		CompressServo.fPosition:= 0;
		CompressServo.fVelocity:= 10; //mm/s
	
		CompressServo.xMoveA:=TRUE;
		StateNext:=5;
	5:	
		IF CompressServo.xInPosition = TRUE THEN
		
			CompressServo.xMoveA := FALSE;
			StateNext:=0;
			axis_ready:=TRUE;
		
		END_IF


	END_CASE

	State:=StateNext;
ELSIF NOT enable THEN
	axis_ready:=FALSE;
	CompressServo.xMoveA := FALSE;
	state:=0;
END_IF
END_METHOD

METHOD _Halt : BOOL
VAR_INPUT
END_VAR
CompressServo.xHalt:=TRUE;
END_METHOD

METHOD _Halt_false : BOOL
VAR_INPUT
END_VAR
CompressServo.xHalt:=FALSE;
END_METHOD

METHOD _Home : BOOL
VAR_INPUT
	
END_VAR


VAR

	
	
END_VAR

VAR_OUTPUT
	
END_VAR
CASE State OF //you are here

0:	
	_ExecutedHome := FALSE;
	CompressServo.fVelocity := ToolPositioningSpeed;
	CompressServo.fAxisAcceleration := ToolPositioningAccel;
	CompressServo.fAxisDeceleration := ToolPositioningAccel;
	CompressServo.fAxisJerk := ToolPositioningJerk;

	IF ixCompressHomeSwitch THEN
		CompressServo.xPositiveDirection := FALSE;
		IF  tickcounter_compress < 10 THEN
			tickcounter_compress := tickcounter_compress + 1;  // can be put in onditional
		
		ELSE
		//IF tickcounter_compress >= 10 THEN
			CompressServo.xMoveV := TRUE;
		END_IF
	ELSE
	
		//CompressServo.xHalt := NOT CompressServo.xHalt;
		CompressServo.xMoveV := FALSE;
		//CompressServo.xHalt := NOT CompressServo.xHalt;
		CompressServo.xHalt := TRUE;
		IF CompressServo.xHalted THEN
			tickcounter_compress:=0;
			StateNext := 5;
		END_IF
	
	END_IF
	
5:
	
	CompressServo.xHalt := FALSE;
	tickcounter_compress := tickcounter_compress + 1;
	IF tickcounter_compress >= 10 THEN
		tickcounter_compress := 0;
		StateNext := 10;
	END_IF
	
10:
	CompressServo.fVelocity := ToolHomingSpeed;
	
	IF NOT ixCompressHomeSwitch THEN
		CompressServo.xPositiveDirection := TRUE;
		IF tickcounter_compress < 10 THEN
			tickcounter_compress := tickcounter_compress + 1;
		ELSE
		//IF tickcounter >= 10 THEN
			CompressServo.xMoveV := TRUE;
		END_IF
	ELSE
		CompressServo.xMoveV := FALSE;
		CompressServo.xHalt := TRUE;
		IF CompressServo.xHalted AND CompressServo.fstandstill THEN
			tickcounter_compress := 0;
			StateNext := 15;
		END_IF
	END_IF

15:
	
	CompressServo.xHalt := FALSE;
	tickcounter_compress := tickcounter_compress + 1;
	IF tickcounter_compress >= 25 THEN
		tickcounter_compress := 0;
		StateNext := 20;
		//Executed := TRUE;
	END_IF	

20:
	CompressServo.fHomeOffset := 0;
	CompressServo.xZero := TRUE;
	StateNext := 25;	
	
25:
	IF CompressServo.xZeroed THEN
		CompressServo.xZero := FALSE;
		_ExecutedHome := TRUE;
		StateNext := 0;
	END_IF

END_CASE

State := StateNext;
END_METHOD

METHOD _Home_without_resetting : BOOL
VAR_INPUT
	enable			:BOOL;
END_VAR


VAR

	
	
END_VAR

VAR_OUTPUT
	
END_VAR

IF enable AND NOT axis_ready THEN
	CASE State OF //you are here

	0:	
		//_ExecutedHome := FALSE;
		CompressServo.fVelocity := ToolPositioningSpeed;
		CompressServo.fAxisAcceleration := ToolPositioningAccel;
		CompressServo.fAxisDeceleration := ToolPositioningAccel;
		CompressServo.fAxisJerk := ToolPositioningJerk;

		IF ixCompressHomeSwitch THEN
			CompressServo.xPositiveDirection := FALSE;
			//IF  tickcounter_compress < 10 THEN
			//	tickcounter_compress := tickcounter_compress + 1;  // can be put in onditional
		
			//ELSE
			//IF tickcounter_compress >= 10 THEN
			CompressServo.xMoveV := TRUE;
			//END_IF
		ELSE
	
			//CompressServo.xHalt := NOT CompressServo.xHalt;
			CompressServo.xMoveV := FALSE;
			//CompressServo.xHalt := NOT CompressServo.xHalt;
			CompressServo.xHalt := TRUE;
			statenext:=5;

	
		END_IF	
	5:
	
		IF CompressServo.xHalted THEN
			//tickcounter_compress:=0;
			CompressServo.xHalt := FALSE;
			StateNext := 10;
		END_IF
	
	10:
		CompressServo.fVelocity := ToolHomingSpeed;
	
		IF NOT ixCompressHomeSwitch THEN
			CompressServo.xPositiveDirection := TRUE;
			//IF tickcounter_compress < 10 THEN
			//	tickcounter_compress := tickcounter_compress + 1;
			//ELSE
			//IF tickcounter >= 10 THEN
			CompressServo.xMoveV := TRUE;
			//END_IF
		ELSE
			CompressServo.xMoveV := FALSE;
			CompressServo.xHalt := TRUE;
			IF CompressServo.xHalted AND CompressServo.fstandstill THEN
				tickcounter_compress := 0;
				StateNext := 15;
			END_IF
		END_IF

	15:
	
		CompressServo.xHalt := FALSE;
		tickcounter_compress := tickcounter_compress + 1;
		IF tickcounter_compress >= 25 THEN
			tickcounter_compress := 0;
			StateNext := 20;
			//Executed := TRUE;
		END_IF	

	20:

		//CompressServo.xZero := FALSE;
		axis_ready := TRUE;
		StateNext := 0;
	

	END_CASE

	State := StateNext;

ELSIF enable = FALSE THEN
	axis_ready:=FALSE;
	CompressServo.xHalt:=FALSE;
	CompressServo.xMoveV:=FALSE;
	state:=0;
	statenext:=0;
END_IF
END_METHOD

METHOD _manuel : BOOL
VAR_INPUT
	enable			:BOOL;
END_VAR
IF enable THEN
	IF NOT compress_settings.minus AND compress_settings.plus (*AND compressservo.xHalted*) THEN
		//CompressServo.xMoveV:=TRUE;
		Compressservo.fVelocity:=compress_settings.speed;
		CompressServo.xPositiveDirection := TRUE;
		CompressServo.xMoveV:=TRUE;
		CompressServo.xHalt:=FALSE;
	
	ELSIF NOT compress_settings.plus AND compress_settings.minus (*AND compressservo.xHalted*) THEN
	
		Compressservo.fVelocity:=compress_settings.speed;
		CompressServo.xPositiveDirection := FALSE;
		CompressServo.xMoveV:=TRUE;
		CompressServo.xHalt:=FALSE;	
	
	ELSIF NOT compress_settings.plus AND NOT compress_settings.minus THEN
	
		CompressServo.xHalt:=TRUE;
		CompressServo.xMoveV:=FALSE;
	
	END_IF
ELSE
	CompressServo.xHalt:=FALSE;
	CompressServo.xMoveV:=FALSE;
END_IF
END_METHOD

METHOD _mc_stop : BOOL
VAR_INPUT
END_VAR
CompressServo.xStop:=TRUE;
END_METHOD

METHOD _Reset
VAR_INPUT
END_VAR
	tickcounter_Compress:=0;
	CompressServoEnable := FALSE;
	CompressServo.xZero := FALSE;
	CompressServo.xMoveV := FALSE;
	CompressServo.xMoveA := FALSE;
	CompressServo.xHalt := FALSE;
	CompressServo.GearIn := FALSE;
	CompressServo.xStop:=FALSE;
	state:=0;
	statenext:=0;
	
	
	axis_ready:=FALSE;
	_ExecutedHome:=FALSE;
	_ExecutedOffset:=FALSE;
	PRG_Machine.reset_rec_old();
	PRG_Machine._debug(enable:=FALSE);
END_METHOD

METHOD _Reset_medium
VAR_INPUT
END_VAR
	tickcounter_Compress:=0;
	CompressServoEnable := FALSE;
	CompressServo.xZero := FALSE;
	CompressServo.xMoveV := FALSE;
	CompressServo.xMoveA := FALSE;
	CompressServo.xHalt := FALSE;
	CompressServo.GearIn := FALSE;
	CompressServo.xStop:=FALSE;
	state:=0;
	statenext:=0;
	
	
	axis_ready:=FALSE;
	PRG_Machine._debug(enable:=FALSE);
END_METHOD

METHOD _retract  : BOOL
VAR_INPUT
	Enable				:BOOL;
	
END_VAR
IF enable AND NOT axis_ready THEN
	CASE State OF
	
	0:	
	
		CompressServo.fPosition:= 0;
		CompressServo.fVelocity:= _Compress_Param.Pusher.Retract_Speed; //mm/s
	
		CompressServo.xMoveA:=TRUE;
		StateNext:=5;
	5:	
		IF CompressServo.xInPosition = TRUE THEN
		
			CompressServo.xMoveA := FALSE;
			StateNext:=0;
			axis_ready:=TRUE;
		
		END_IF


	END_CASE

	State:=StateNext;
ELSIF NOT enable THEN
	axis_ready:=FALSE;
	CompressServo.xMoveA := FALSE;
	state:=0;
END_IF
END_METHOD

METHOD _Soft_Reset
VAR_INPUT
END_VAR

tickcounter_Compress:=0;
CompressServo.xZero := FALSE;
CompressServo.xMoveV := FALSE;
CompressServo.xMoveA := FALSE;
CompressServo.xHalt := FALSE;
CompressServo.GearIn := FALSE;
CompressServo.xStop:=FALSE;
state:=0;
statenext:=0;

axis_ready:=FALSE;
PRG_Machine._debug(enable:=FALSE);
END_METHOD

METHOD _Update
VAR_INPUT
END_VAR
CompressServo(
	xEnable:= CompressServoEnable, 
	xZero:= , 
	xMoveR:= , 
	xMoveA:= , 
	xMoveV:= , 
	xPositiveDirection:= , 
	fDistance:= , 
	fPosition:= , 
	fVelocity:= , 
	xStop:= , 
	xHome:= , 
	xHomeFlag:= , 
	homePosition:=0,
	fActualPosition=> , 
	fActualVelocity=> , 
	fActModuloPos=> , 
	xEnabled=> CompressServoEnabled, 
	xMoveComplete=> , 
	xInPosition=> , 
	xAtSpeed=> , 
	xStopped=> , 
	xHomed=> ,
	errorID=> CompressServoErrorID, 
	Axis:= CompressAxis );
END_METHOD

PROPERTY Compress_Param : recipe
GET
Compress_param := _Compress_Param;
END_GET
SET
_Compress_param := Compress_Param;
END_SET
END_PROPERTY

PROPERTY HomeExecuted : BOOL
GET
HomeExecuted := _ExecutedHome;
END_GET
SET
_ExecutedHome := HomeExecuted;
END_SET
END_PROPERTY

METHOD Offset
VAR_INPUT
	Enable				:BOOL;
END_VAR

IF enable AND NOT axis_ready THEN	
	CASE State OF
	0:	
		_ExecutedOffset:=FALSE;
		CompressServo.fPosition:= _Compress_Param.Other.Compress_Home_Offset - PRG_Machine.rec_old.other.Compress_home_offset;
		CompressServo.fVelocity:= 20; //mm/s
	
		IF CompressServo.fPosition<>0 THEN
			CompressServo.xMoveA:=TRUE;
			StateNext:=5;
		ELSE
			_ExecutedOffset:=TRUE;
		END_IF
	
		//StateNext:=5;
	5:	
		IF CompressServo.xInPosition AND compressservo.fstandstill = TRUE THEN
			
			CompressServo.xMoveA := FALSE;
			StateNext:=7;
			//_ExecutedOffset:=TRUE;
		
		END_IF
	
	7:

		tickcounter_compress := tickcounter_compress + 1;
		IF tickcounter_compress >= 25 THEN
			tickcounter_compress := 0;
			StateNext := 10;
			//Executed := TRUE;
		END_IF	
	
	10:
	
		compressServo.fHomeOffset := 0;
		compressServo.xZero := TRUE;
		StateNext := 15;	
	
	15:
		IF compressServo.xZeroed THEN
			compressServo.xZero := FALSE;
			_ExecutedOffset:=TRUE;
			axis_ready:=TRUE;
			StateNext := 0;
		END_IF

	END_CASE

	State:=StateNext;
	
ELSIF NOT enable THEN 
	axis_ready:=FALSE;
	compressServo.xZero := FALSE;
	StateNext := 0;
END_IF
END_METHOD

PROPERTY OffsetExecuted : BOOL
GET
OffsetExecuted := _ExecutedOffset;
END_GET
SET
_ExecutedOffset := OffsetExecuted;
END_SET
END_PROPERTY

PROPERTY Stage1Executed : BOOL
GET
Stage1Executed := _ExecutedStage1;
END_GET
SET
_ExecutedStage1 := Stage1Executed;
END_SET
END_PROPERTY

PROPERTY Stage5Executed : BOOL
GET
Stage5Executed := _ExecutedStage5;
END_GET
SET
_ExecutedStage5 := Stage5Executed;
END_SET
END_PROPERTY

END_FUNCTION_BLOCK

// ---- Classes/Shield/FB_Shield.TcPOU
FUNCTION_BLOCK FB_Shield
VAR_INPUT
END_VAR
VAR_OUTPUT
	Axis_ready					:BOOL:=FALSE;
END_VAR
VAR

ShieldServo: 		FB_AxisControl;

_Shield_param				:recipe;

distance1:					LREAL:=67;




ToolPositioningSpeed	: LREAL := 20;
ToolPositioningAccel	: LREAL := 100;
ToolPositioningJerk		: LREAL := 1000;
ToolHomingSpeed			: LREAL := 2;

ShieldServoEnable:  BOOL;
ShieldServoEnabled: BOOL;

_ExecutedHome				:BOOL:=FALSE;
_ExecutedStage2 			:BOOL:=FALSE;
_ExecutedStage3				:BOOL:=FALSE;
_ExecutedOffset				:BOOL:=FALSE;

tickcounter_shield: 		INT :=0;
State: 						INT:= 0;
StateNext: 					INT:= 0;

END_VAR

METHOD _absolute_move : BOOL
VAR_INPUT
	Enable				:BOOL;
	Stage				:INT;
END_VAR
IF Enable AND NOT Axis_ready THEN
	CASE State OF
	
	0:	
		
		ShieldServo.fPosition:= _Shield_Param.Shield.Distance[Stage];
		ShieldServo.fVelocity:= _Shield_Param.Shield.Speed[Stage]; //mm/s
	
	
		ShieldServo.xMoveA:=TRUE;
	
	
		StateNext:=5;
	5:	
		IF ShieldServo.xInPosition = TRUE THEN
		
			ShieldServo.xMoveA := FALSE;
			StateNext:=0;
			axis_ready:=TRUE;
		
		
		END_IF


	END_CASE

	State:=StateNext;
ELSIF NOT enable THEN
	axis_ready:=FALSE;
	ShieldServo.xMoveA := FALSE;
	state:=0;
END_IF
END_METHOD

METHOD _Enable 
VAR_INPUT
END_VAR

ShieldServoEnable := TRUE;
END_METHOD

METHOD _force_home  : BOOL
VAR_INPUT
	Enable				:BOOL;
	
END_VAR
IF enable AND NOT axis_ready THEN
	CASE State OF
	
	0:	
	
		ShieldServo.fPosition:= 0;
		ShieldServo.fVelocity:= 10; //mm/s
	
		ShieldServo.xMoveA:=TRUE;
		StateNext:=5;
	5:	
		IF ShieldServo.xInPosition = TRUE THEN
		
			ShieldServo.xMoveA := FALSE;
			StateNext:=0;
			axis_ready:=TRUE;
		
		END_IF


	END_CASE

	State:=StateNext;
ELSIF enable = FALSE THEN
	axis_ready:=FALSE;
	ShieldServo.xMoveA := FALSE;
	state:=0;
END_IF
END_METHOD

METHOD _Halt : BOOL
VAR_INPUT
END_VAR
ShieldServo.xHalt:=TRUE;
END_METHOD

METHOD _Halt_false : BOOL
VAR_INPUT
END_VAR
ShieldServo.xHalt:=FALSE;
END_METHOD

METHOD _Home 
VAR_INPUT
	
END_VAR


VAR



END_VAR

VAR_OUTPUT
	
END_VAR





CASE State OF //you are here



0:	
	_ExecutedHome := FALSE;
	ShieldServo.fVelocity := ToolPositioningSpeed;
	ShieldServo.fAxisAcceleration := ToolPositioningAccel;
	ShieldServo.fAxisDeceleration := ToolPositioningAccel;
	ShieldServo.fAxisJerk := ToolPositioningJerk;

	IF ixShieldHomeSwitch THEN
		ShieldServo.xPositiveDirection := FALSE;
		IF  tickcounter_shield < 10 THEN
			tickcounter_shield := tickcounter_shield + 1;  // can be put in onditional
		
		ELSE
		//IF tickcounter_compress >= 10 THEN
			ShieldServo.xMoveV := TRUE;
		END_IF
	ELSE
	
		//CompressServo.xHalt := NOT CompressServo.xHalt;
		ShieldServo.xMoveV := FALSE;
		//CompressServo.xHalt := NOT CompressServo.xHalt;
		ShieldServo.xHalt := TRUE;
		IF ShieldServo.xHalted THEN
			tickcounter_shield:=0;
			StateNext := 5;
		END_IF
	
	END_IF
	
5:
	
	ShieldServo.xHalt := FALSE;
	tickcounter_shield := tickcounter_shield + 1;
	IF tickcounter_shield >= 10 THEN
		tickcounter_shield := 0;
		StateNext := 10;
	END_IF
	
10:
	ShieldServo.fVelocity := ToolHomingSpeed;
	
	IF NOT ixShieldHomeSwitch THEN
		ShieldServo.xPositiveDirection := TRUE;
		IF tickcounter_shield < 10 THEN
			tickcounter_shield := tickcounter_shield + 1;
		ELSE
		//IF tickcounter >= 10 THEN
			shieldServo.xMoveV := TRUE;
		END_IF
	ELSE
		shieldServo.xMoveV := FALSE;
		shieldServo.xHalt := TRUE;
		IF shieldServo.xHalted AND shieldservo.fstandstill THEN
			tickcounter_shield := 0;
			StateNext := 15;
		END_IF
	END_IF

15:
	
	shieldServo.xHalt := FALSE;
	tickcounter_shield := tickcounter_shield + 1;
	IF tickcounter_shield >= 25 THEN
		tickcounter_shield := 0;
		StateNext := 20;
		//Executed := TRUE;
	END_IF
20:
	shieldServo.fHomeOffset := 0;
	shieldServo.xZero := TRUE;
	StateNext := 25;	
	
25:
	IF shieldServo.xZeroed THEN
		shieldServo.xZero := FALSE;
		_ExecutedHome := TRUE;
		StateNext := 0;
	END_IF
	

END_CASE

State := StateNext;
END_METHOD

METHOD _mc_stop : BOOL
VAR_INPUT
END_VAR
ShieldServo.xStop:=TRUE;
END_METHOD

METHOD _Reset
VAR_INPUT
END_VAR
	tickcounter_Shield:=0;
	ShieldServoEnable := FALSE;
	ShieldServo.xZero := FALSE;
	ShieldServo.xMoveV := FALSE;
	ShieldServo.xMoveA := FALSE;
	ShieldServo.xHalt := FALSE;
	ShieldServo.GearIn := FALSE;
	ShieldServo.xStop:=FALSE;
	state:=0;
	statenext:=0;
	
	
	axis_ready:=FALSE;
	_ExecutedHome:=FALSE;
	_ExecutedOffset:=FALSE;
	PRG_Machine.reset_rec_old();
	PRG_Machine._debug(enable:=FALSE);
END_METHOD

METHOD _Reset_medium
VAR_INPUT
END_VAR
	tickcounter_Shield:=0;
	ShieldServoEnable := FALSE;
	ShieldServo.xZero := FALSE;
	ShieldServo.xMoveV := FALSE;
	ShieldServo.xMoveA := FALSE;
	ShieldServo.xHalt := FALSE;
	ShieldServo.GearIn := FALSE;
	ShieldServo.xStop:=FALSE;
	state:=0;
	statenext:=0;
	
	axis_ready:=FALSE;
	PRG_Machine._debug(enable:=FALSE);
END_METHOD

METHOD _retract  : BOOL
VAR_INPUT
	Enable				:BOOL;
	
END_VAR
IF enable AND NOT axis_ready THEN
	CASE State OF
	
	0:	
	
		ShieldServo.fPosition:= 0;
		ShieldServo.fVelocity:= _Shield_Param.Pusher.Retract_Speed; //mm/s
	
		ShieldServo.xMoveA:=TRUE;
		StateNext:=5;
	5:	
		IF ShieldServo.xInPosition = TRUE THEN
		
			ShieldServo.xMoveA := FALSE;
			StateNext:=0;
			axis_ready:=TRUE;
		
		END_IF


	END_CASE

	State:=StateNext;
ELSIF enable = FALSE THEN
	axis_ready:=FALSE;
	ShieldServo.xMoveA := FALSE;
	state:=0;
END_IF
END_METHOD

METHOD _Soft_Reset
VAR_INPUT
END_VAR

tickcounter_Shield:=0;
ShieldServo.xZero := FALSE;
ShieldServo.xMoveV := FALSE;
ShieldServo.xMoveA := FALSE;
ShieldServo.xHalt := FALSE;
ShieldServo.GearIn := FALSE;
ShieldServo.xStop:=FALSE;
state:=0;
statenext:=0;

axis_ready:=FALSE;
PRG_Machine._debug(enable:=FALSE);
END_METHOD

METHOD _Update
VAR_INPUT
END_VAR
ShieldServo(
	xEnable:= ShieldServoEnable, 
	xZero:= , 
	xMoveR:= , 
	xMoveA:= , 
	xMoveV:= , 
	xPositiveDirection:= , 
	fDistance:= , 
	fPosition:= , 
	fVelocity:= , 
	xStop:= , 
	xHome:= , 
	xHomeFlag:= , 
	homePosition:=0,
	fActualPosition=> , 
	fActualVelocity=> , 
	fActModuloPos=> , 
	xEnabled=> ShieldServoEnabled, 
	xMoveComplete=> , 
	xInPosition=> , 
	xAtSpeed=> , 
	xStopped=> , 
	xHomed=> ,
	errorID=> ShieldServoErrorID, 
	Axis:= ShieldAxis );
END_METHOD

PROPERTY HomeExecuted : BOOL;
GET
HomeExecuted := _ExecutedHome;
END_GET
SET
_ExecutedHome := HomeExecuted;
END_SET
END_PROPERTY

METHOD Offset
VAR_INPUT
	Enable				:BOOL;
END_VAR

IF enable AND NOT axis_ready THEN	
	CASE State OF
	0:	
		_ExecutedOffset:=FALSE;
		ShieldServo.fPosition:= _Shield_Param.Other.Shield_Home_Offset-PRG_Machine.rec_old.other.shield_home_offset;
		ShieldServo.fVelocity:= 20; //mm/s
	
		IF ShieldServo.fPosition<>0 THEN
			ShieldServo.xMoveA:=TRUE;
			StateNext:=5;
		ELSE
			_ExecutedOffset:=TRUE;
		END_IF
	
		//StateNext:=5;
	5:	
		IF ShieldServo.xInPosition = TRUE AND ShieldServo.fstandstill THEN
			
			ShieldServo.xMoveA := FALSE;
			StateNext:=7;
			//_ExecutedOffset:=TRUE;
		
		END_IF
		
	7:
		tickcounter_shield:=tickcounter_shield+1;
		IF tickcounter_shield >= 25 THEN
			tickcounter_shield := 0;
			StateNext := 10;
			//Executed := TRUE;
		END_IF
		
	10:
	
		ShieldServo.fHomeOffset := 0;
		ShieldServo.xZero := TRUE;
		StateNext := 15;	
	
	15:
		IF shieldServo.xZeroed THEN
			shieldServo.xZero := FALSE;
			_ExecutedOffset:=TRUE;
			axis_ready:=TRUE;
			StateNext := 0;
		END_IF

	END_CASE

	State:=StateNext;
	
ELSIF NOT enable THEN 
	axis_ready:=FALSE;
	ShieldServo.xZero := FALSE;
	
	StateNext := 0;
END_IF
END_METHOD

PROPERTY OffsetExecuted : BOOL
GET
OffsetExecuted := _ExecutedOffset;
END_GET
SET
_ExecutedOffset := OffsetExecuted;
END_SET
END_PROPERTY

PROPERTY Shield_Param : recipe
GET
Shield_param := _Shield_Param;
END_GET
SET
_Shield_param := Shield_Param;
END_SET
END_PROPERTY

PROPERTY Stage2Executed : BOOL
GET
Stage2Executed := _ExecutedStage2;
END_GET
SET
_ExecutedStage2 := Stage2Executed;
END_SET
END_PROPERTY

PROPERTY Stage3Executed : BOOL
GET
Stage3Executed := _ExecutedStage3;
END_GET
SET
_ExecutedStage3 := Stage3Executed;
END_SET
END_PROPERTY

END_FUNCTION_BLOCK

// ---- POUs/Config_Slow.TcPOU
PROGRAM Config_Slow
VAR
	//temp					:INT;
	//temp_load				:INT :=1;
	//temp_save				:INT :=0;
	Once					:BOOL :=TRUE;
	juan					:INT;
	//saving_config			:BOOL :=FALSE;
	//config_status			:BOOL :=FALSE;
	config_count			:INT;		
END_VAR


IF Clock.DateTimeInitialised THEN
	
	FOR juan := 1 TO config_speed DO
		Config.Update();
	END_FOR

	
	
	load_config();
	
	IF config.Initialised() THEN
		save_config();	
	END_IF

END_IF

METHOD load_config : BOOL
VAR_INPUT
END_VAR
(*//IF once =TRUE THEN
	IF Config.Initialised(temp_load) = FALSE THEN
		Config.Update(temp_load);


	ELSIF temp_load = 11 THEN
		Message:='Data Loaded';
		Once:=FALSE;
	ELSE
		Config.Update(temp_load);
		Config.Update(temp_load);
		temp_load:=temp_load+1;
	END_IF
//END_IF
*)	
//2500
//Config.Update(1);
//Config.Update(2);
//Config.Update(3);
//Config.Update(4);
//Config.Update(5);
//Config.Update(6);
//Config.Update(7);
//Config.Update(8);
//Config.Update(9);
//Config.Update(10);
//Config.Update(11);

IF once AND config.Initialised() THEN
	once:=FALSE;
	IF language.english THEN
		Message:='Data loaded';
	ELSE
		Message:='Dados carregados';
	END_IF
END_IF


(*
IF config_count = 1000 THEN
	config_count:=0;
	IF temp_load = 11 THEN
		temp_load:=0;
	END_IF 
	temp_load:=temp_load+1;
END_IF
*)
END_METHOD

METHOD save_config : BOOL
VAR_INPUT
END_VAR

	
IF Config_Request= TRUE THEN
	Config_Request:=FALSE;

	config_count:=0;
	//temp_save:=temp_save+1;
		
END_IF

config_count:=config_count+config_speed;

IF config_count > 7000 THEN
	config_count := 0;
	IF configuring THEN
		Message:=Config_Message;
		configuring:=FALSE;
	END_IF
	
END_IF
END_METHOD

END_PROGRAM

// ---- Classes/Config/TConfig.TcPOU
FUNCTION_BLOCK TConfig
VAR
    Recipe_mem_name 						AT %MD0: STRING(20);

	
	Rec_Name_1								AT %MD0 :UDINT;
	Rec_Name_2								AT %MD1 :UDINT;
	Rec_Name_3								AT %MD2 :UDINT;
	Rec_Name_4								AT %MD3 :UDINT;
	Rec_Name_5								AT %MD4 :UDINT;

	
	PersistentData 						: TPersistentData;
	
    
	ConfigData							:  TConfigData;

		
END_VAR

METHOD CopyConfigRecipiesToGlobal : BOOL
VAR_INPUT

END_VAR

limits_save.max_limit_Compress:=ConfigData.con_max_limit_Compress;
Limits_save.max_limit_Pusher:=ConfigData.con_max_limit_Pusher;
Limits_save.max_limit_Shield:=ConfigData.con_max_limit_Shield;
Limits_save.max_pusher_shield_diff:=ConfigData.con_max_pusher_shield_diff;	
Limits_save.max_torque:=ConfigData.con_max_torque;

//1
Rec_Name_1:=ConfigData.rec1_Name_1;								
Rec_Name_2:=ConfigData.rec1_Name_2;								
Rec_Name_3:=ConfigData.rec1_Name_3;								
Rec_Name_4:=ConfigData.rec1_Name_4;								
Rec_Name_5:=ConfigData.rec1_Name_5;
List_of_Recipes[1].Name:=Recipe_mem_name;

List_of_Recipes[1].Shield.Retract_Speed :=ConfigData.rec1_Shield_Retract_Speed;
List_of_Recipes[1].Shield.Speed[1] := ConfigData.rec1_Shield_Speed_1;
List_of_Recipes[1].Shield.Speed[2] := ConfigData.rec1_Shield_Speed_2;
List_of_Recipes[1].Shield.Speed[3] := ConfigData.rec1_Shield_Speed_3;
List_of_Recipes[1].Shield.Speed[4] := ConfigData.rec1_Shield_Speed_4;
List_of_Recipes[1].Shield.Speed[5] := ConfigData.rec1_Shield_Speed_5;
List_of_Recipes[1].Shield.Speed[6] := ConfigData.rec1_Shield_Speed_6;
List_of_Recipes[1].Shield.distance[1] := ConfigData.rec1_Shield_distance_1;
List_of_Recipes[1].Shield.distance[2] := ConfigData.rec1_Shield_distance_2;
List_of_Recipes[1].Shield.distance[3] := ConfigData.rec1_Shield_distance_3;
List_of_Recipes[1].Shield.distance[4] := ConfigData.rec1_Shield_distance_4;
List_of_Recipes[1].Shield.distance[5] := ConfigData.rec1_Shield_distance_5;
List_of_Recipes[1].Shield.distance[6] := ConfigData.rec1_Shield_distance_6;


List_of_Recipes[1].Pusher.Retract_Speed :=ConfigData.rec1_Pusher_Retract_Speed;
List_of_Recipes[1].Pusher.Speed[1] := ConfigData.rec1_Pusher_Speed_1;
List_of_Recipes[1].Pusher.Speed[2] := ConfigData.rec1_Pusher_Speed_2;
List_of_Recipes[1].Pusher.Speed[3] := ConfigData.rec1_Pusher_Speed_3;
List_of_Recipes[1].Pusher.Speed[4] := ConfigData.rec1_Pusher_Speed_4;
List_of_Recipes[1].Pusher.Speed[5] := ConfigData.rec1_Pusher_Speed_5;
List_of_Recipes[1].Pusher.Speed[6] := ConfigData.rec1_Pusher_Speed_6;
List_of_Recipes[1].Pusher.distance[1] := ConfigData.rec1_Pusher_distance_1;
List_of_Recipes[1].Pusher.distance[2] := ConfigData.rec1_Pusher_distance_2;
List_of_Recipes[1].Pusher.distance[3] := ConfigData.rec1_Pusher_distance_3;
List_of_Recipes[1].Pusher.distance[4] := ConfigData.rec1_Pusher_distance_4;
List_of_Recipes[1].Pusher.distance[5] := ConfigData.rec1_Pusher_distance_5;
List_of_Recipes[1].Pusher.distance[6] := ConfigData.rec1_Pusher_distance_6;

List_of_Recipes[1].Compress.Initial_Distance := ConfigData.rec1_Compress_Initial_Distance;
List_of_Recipes[1].Compress.Initial_Speed := ConfigData.rec1_Compress_Initial_Speed;
List_of_Recipes[1].Compress.relax_Distance := ConfigData.rec1_Compress_Relax_Distance;
List_of_Recipes[1].Compress.retract_speed := ConfigData.rec1_Compress_retract_speed;

List_of_Recipes[1].Clamp.Release_Instance:=ConfigData.rec1_Clamp_Release_Instance;

List_of_Recipes[1].Other.Compress_Home_Offset:=ConfigData.rec1_Other_Compress_Home_Offset;
List_of_Recipes[1].Other.Shield_Home_Offset:=ConfigData.rec1_Other_Shield_Home_Offset;
List_of_Recipes[1].Other.Pusher_Home_Offset:=ConfigData.rec1_Other_Pusher_Home_Offset;

List_of_Recipes[1].Memory_Free:=LREAL_TO_BOOL(ConfigData.rec1_Memory_Free);

//2
Rec_Name_1:=ConfigData.rec2_Name_1;								
Rec_Name_2:=ConfigData.rec2_Name_2;								
Rec_Name_3:=ConfigData.rec2_Name_3;								
Rec_Name_4:=ConfigData.rec2_Name_4;								
Rec_Name_5:=ConfigData.rec2_Name_5;
List_of_Recipes[2].Name:=Recipe_mem_name;

List_of_Recipes[2].Shield.Retract_Speed :=ConfigData.rec2_Shield_Retract_Speed;
List_of_Recipes[2].Shield.Speed[1] := ConfigData.rec2_Shield_Speed_1;
List_of_Recipes[2].Shield.Speed[2] := ConfigData.rec2_Shield_Speed_2;
List_of_Recipes[2].Shield.Speed[3] := ConfigData.rec2_Shield_Speed_3;
List_of_Recipes[2].Shield.Speed[4] := ConfigData.rec2_Shield_Speed_4;
List_of_Recipes[2].Shield.Speed[5] := ConfigData.rec2_Shield_Speed_5;
List_of_Recipes[2].Shield.Speed[6] := ConfigData.rec2_Shield_Speed_6;
List_of_Recipes[2].Shield.distance[1] := ConfigData.rec2_Shield_distance_1;
List_of_Recipes[2].Shield.distance[2] := ConfigData.rec2_Shield_distance_2;
List_of_Recipes[2].Shield.distance[3] := ConfigData.rec2_Shield_distance_3;
List_of_Recipes[2].Shield.distance[4] := ConfigData.rec2_Shield_distance_4;
List_of_Recipes[2].Shield.distance[5] := ConfigData.rec2_Shield_distance_5;
List_of_Recipes[2].Shield.distance[6] := ConfigData.rec2_Shield_distance_6;


List_of_Recipes[2].Pusher.Retract_Speed :=ConfigData.rec2_Pusher_Retract_Speed;
List_of_Recipes[2].Pusher.Speed[1] := ConfigData.rec2_Pusher_Speed_1;
List_of_Recipes[2].Pusher.Speed[2] := ConfigData.rec2_Pusher_Speed_2;
List_of_Recipes[2].Pusher.Speed[3] := ConfigData.rec2_Pusher_Speed_3;
List_of_Recipes[2].Pusher.Speed[4] := ConfigData.rec2_Pusher_Speed_4;
List_of_Recipes[2].Pusher.Speed[5] := ConfigData.rec2_Pusher_Speed_5;
List_of_Recipes[2].Pusher.Speed[6] := ConfigData.rec2_Pusher_Speed_6;
List_of_Recipes[2].Pusher.distance[1] := ConfigData.rec2_Pusher_distance_1;
List_of_Recipes[2].Pusher.distance[2] := ConfigData.rec2_Pusher_distance_2;
List_of_Recipes[2].Pusher.distance[3] := ConfigData.rec2_Pusher_distance_3;
List_of_Recipes[2].Pusher.distance[4] := ConfigData.rec2_Pusher_distance_4;
List_of_Recipes[2].Pusher.distance[5] := ConfigData.rec2_Pusher_distance_5;
List_of_Recipes[2].Pusher.distance[6] := ConfigData.rec2_Pusher_distance_6;

List_of_Recipes[2].Compress.Initial_Distance := ConfigData.rec2_Compress_Initial_Distance;
List_of_Recipes[2].Compress.Initial_Speed := ConfigData.rec2_Compress_Initial_Speed;
List_of_Recipes[2].Compress.relax_Distance := ConfigData.rec2_Compress_Relax_Distance;
List_of_Recipes[2].Compress.retract_speed := ConfigData.rec2_Compress_retract_speed;

List_of_Recipes[2].Clamp.Release_Instance:=ConfigData.rec2_Clamp_Release_Instance;

List_of_Recipes[2].Other.Compress_Home_Offset:=ConfigData.rec2_Other_Compress_Home_Offset;
List_of_Recipes[2].Other.Shield_Home_Offset:=ConfigData.rec2_Other_Shield_Home_Offset;
List_of_Recipes[2].Other.Pusher_Home_Offset:=ConfigData.rec2_Other_Pusher_Home_Offset;

List_of_Recipes[2].Memory_Free:=LREAL_TO_BOOL(ConfigData.rec2_Memory_Free);

//3
Rec_Name_1:=ConfigData.rec3_Name_1;								
Rec_Name_2:=ConfigData.rec3_Name_2;								
Rec_Name_3:=ConfigData.rec3_Name_3;								
Rec_Name_4:=ConfigData.rec3_Name_4;								
Rec_Name_5:=ConfigData.rec3_Name_5;
List_of_Recipes[3].Name:=Recipe_mem_name;

List_of_Recipes[3].Shield.Retract_Speed :=ConfigData.rec3_Shield_Retract_Speed;
List_of_Recipes[3].Shield.Speed[1] := ConfigData.rec3_Shield_Speed_1;
List_of_Recipes[3].Shield.Speed[2] := ConfigData.rec3_Shield_Speed_2;
List_of_Recipes[3].Shield.Speed[3] := ConfigData.rec3_Shield_Speed_3;
List_of_Recipes[3].Shield.Speed[4] := ConfigData.rec3_Shield_Speed_4;
List_of_Recipes[3].Shield.Speed[5] := ConfigData.rec3_Shield_Speed_5;
List_of_Recipes[3].Shield.Speed[6] := ConfigData.rec3_Shield_Speed_6;
List_of_Recipes[3].Shield.distance[1] := ConfigData.rec3_Shield_distance_1;
List_of_Recipes[3].Shield.distance[2] := ConfigData.rec3_Shield_distance_2;
List_of_Recipes[3].Shield.distance[3] := ConfigData.rec3_Shield_distance_3;
List_of_Recipes[3].Shield.distance[4] := ConfigData.rec3_Shield_distance_4;
List_of_Recipes[3].Shield.distance[5] := ConfigData.rec3_Shield_distance_5;
List_of_Recipes[3].Shield.distance[6] := ConfigData.rec3_Shield_distance_6;


List_of_Recipes[3].Pusher.Retract_Speed :=ConfigData.rec3_Pusher_Retract_Speed;
List_of_Recipes[3].Pusher.Speed[1] := ConfigData.rec3_Pusher_Speed_1;
List_of_Recipes[3].Pusher.Speed[2] := ConfigData.rec3_Pusher_Speed_2;
List_of_Recipes[3].Pusher.Speed[3] := ConfigData.rec3_Pusher_Speed_3;
List_of_Recipes[3].Pusher.Speed[4] := ConfigData.rec3_Pusher_Speed_4;
List_of_Recipes[3].Pusher.Speed[5] := ConfigData.rec3_Pusher_Speed_5;
List_of_Recipes[3].Pusher.Speed[6] := ConfigData.rec3_Pusher_Speed_6;
List_of_Recipes[3].Pusher.distance[1] := ConfigData.rec3_Pusher_distance_1;
List_of_Recipes[3].Pusher.distance[2] := ConfigData.rec3_Pusher_distance_2;
List_of_Recipes[3].Pusher.distance[3] := ConfigData.rec3_Pusher_distance_3;
List_of_Recipes[3].Pusher.distance[4] := ConfigData.rec3_Pusher_distance_4;
List_of_Recipes[3].Pusher.distance[5] := ConfigData.rec3_Pusher_distance_5;
List_of_Recipes[3].Pusher.distance[6] := ConfigData.rec3_Pusher_distance_6;

List_of_Recipes[3].Compress.Initial_Distance := ConfigData.rec3_Compress_Initial_Distance;
List_of_Recipes[3].Compress.Initial_Speed := ConfigData.rec3_Compress_Initial_Speed;
List_of_Recipes[3].Compress.relax_Distance := ConfigData.rec3_Compress_Relax_Distance;
List_of_Recipes[3].Compress.retract_speed := ConfigData.rec3_Compress_retract_speed;

List_of_Recipes[3].Clamp.Release_Instance:=ConfigData.rec3_Clamp_Release_Instance;

List_of_Recipes[3].Other.Compress_Home_Offset:=ConfigData.rec3_Other_Compress_Home_Offset;
List_of_Recipes[3].Other.Shield_Home_Offset:=ConfigData.rec3_Other_Shield_Home_Offset;
List_of_Recipes[3].Other.Pusher_Home_Offset:=ConfigData.rec3_Other_Pusher_Home_Offset;

List_of_Recipes[3].Memory_Free:=LREAL_TO_BOOL(ConfigData.rec3_Memory_Free);

//4
Rec_Name_1:=ConfigData.rec4_Name_1;								
Rec_Name_2:=ConfigData.rec4_Name_2;								
Rec_Name_3:=ConfigData.rec4_Name_3;								
Rec_Name_4:=ConfigData.rec4_Name_4;								
Rec_Name_5:=ConfigData.rec4_Name_5;
List_of_Recipes[4].Name:=Recipe_mem_name;

List_of_Recipes[4].Shield.Retract_Speed :=ConfigData.rec4_Shield_Retract_Speed;
List_of_Recipes[4].Shield.Speed[1] := ConfigData.rec4_Shield_Speed_1;
List_of_Recipes[4].Shield.Speed[2] := ConfigData.rec4_Shield_Speed_2;
List_of_Recipes[4].Shield.Speed[3] := ConfigData.rec4_Shield_Speed_3;
List_of_Recipes[4].Shield.Speed[4] := ConfigData.rec4_Shield_Speed_4;
List_of_Recipes[4].Shield.Speed[5] := ConfigData.rec4_Shield_Speed_5;
List_of_Recipes[4].Shield.Speed[6] := ConfigData.rec4_Shield_Speed_6;
List_of_Recipes[4].Shield.distance[1] := ConfigData.rec4_Shield_distance_1;
List_of_Recipes[4].Shield.distance[2] := ConfigData.rec4_Shield_distance_2;
List_of_Recipes[4].Shield.distance[3] := ConfigData.rec4_Shield_distance_3;
List_of_Recipes[4].Shield.distance[4] := ConfigData.rec4_Shield_distance_4;
List_of_Recipes[4].Shield.distance[5] := ConfigData.rec4_Shield_distance_5;
List_of_Recipes[4].Shield.distance[6] := ConfigData.rec4_Shield_distance_6;


List_of_Recipes[4].Pusher.Retract_Speed :=ConfigData.rec4_Pusher_Retract_Speed;
List_of_Recipes[4].Pusher.Speed[1] := ConfigData.rec4_Pusher_Speed_1;
List_of_Recipes[4].Pusher.Speed[2] := ConfigData.rec4_Pusher_Speed_2;
List_of_Recipes[4].Pusher.Speed[3] := ConfigData.rec4_Pusher_Speed_3;
List_of_Recipes[4].Pusher.Speed[4] := ConfigData.rec4_Pusher_Speed_4;
List_of_Recipes[4].Pusher.Speed[5] := ConfigData.rec4_Pusher_Speed_5;
List_of_Recipes[4].Pusher.Speed[6] := ConfigData.rec4_Pusher_Speed_6;
List_of_Recipes[4].Pusher.distance[1] := ConfigData.rec4_Pusher_distance_1;
List_of_Recipes[4].Pusher.distance[2] := ConfigData.rec4_Pusher_distance_2;
List_of_Recipes[4].Pusher.distance[3] := ConfigData.rec4_Pusher_distance_3;
List_of_Recipes[4].Pusher.distance[4] := ConfigData.rec4_Pusher_distance_4;
List_of_Recipes[4].Pusher.distance[5] := ConfigData.rec4_Pusher_distance_5;
List_of_Recipes[4].Pusher.distance[6] := ConfigData.rec4_Pusher_distance_6;

List_of_Recipes[4].Compress.Initial_Distance := ConfigData.rec4_Compress_Initial_Distance;
List_of_Recipes[4].Compress.Initial_Speed := ConfigData.rec4_Compress_Initial_Speed;
List_of_Recipes[4].Compress.relax_Distance := ConfigData.rec4_Compress_Relax_Distance;
List_of_Recipes[4].Compress.retract_speed := ConfigData.rec4_Compress_retract_speed;

List_of_Recipes[4].Clamp.Release_Instance:=ConfigData.rec4_Clamp_Release_Instance;

List_of_Recipes[4].Other.Compress_Home_Offset:=ConfigData.rec4_Other_Compress_Home_Offset;
List_of_Recipes[4].Other.Shield_Home_Offset:=ConfigData.rec4_Other_Shield_Home_Offset;
List_of_Recipes[4].Other.Pusher_Home_Offset:=ConfigData.rec4_Other_Pusher_Home_Offset;

List_of_Recipes[4].Memory_Free:=LREAL_TO_BOOL(ConfigData.rec4_Memory_Free);		

//5
Rec_Name_1:=ConfigData.rec5_Name_1;								
Rec_Name_2:=ConfigData.rec5_Name_2;								
Rec_Name_3:=ConfigData.rec5_Name_3;								
Rec_Name_4:=ConfigData.rec5_Name_4;								
Rec_Name_5:=ConfigData.rec5_Name_5;
List_of_Recipes[5].Name:=Recipe_mem_name;

List_of_Recipes[5].Shield.Retract_Speed :=ConfigData.rec5_Shield_Retract_Speed;
List_of_Recipes[5].Shield.Speed[1] := ConfigData.rec5_Shield_Speed_1;
List_of_Recipes[5].Shield.Speed[2] := ConfigData.rec5_Shield_Speed_2;
List_of_Recipes[5].Shield.Speed[3] := ConfigData.rec5_Shield_Speed_3;
List_of_Recipes[5].Shield.Speed[4] := ConfigData.rec5_Shield_Speed_4;
List_of_Recipes[5].Shield.Speed[5] := ConfigData.rec5_Shield_Speed_5;
List_of_Recipes[5].Shield.Speed[6] := ConfigData.rec5_Shield_Speed_6;
List_of_Recipes[5].Shield.distance[1] := ConfigData.rec5_Shield_distance_1;
List_of_Recipes[5].Shield.distance[2] := ConfigData.rec5_Shield_distance_2;
List_of_Recipes[5].Shield.distance[3] := ConfigData.rec5_Shield_distance_3;
List_of_Recipes[5].Shield.distance[4] := ConfigData.rec5_Shield_distance_4;
List_of_Recipes[5].Shield.distance[5] := ConfigData.rec5_Shield_distance_5;
List_of_Recipes[5].Shield.distance[6] := ConfigData.rec5_Shield_distance_6;


List_of_Recipes[5].Pusher.Retract_Speed :=ConfigData.rec5_Pusher_Retract_Speed;
List_of_Recipes[5].Pusher.Speed[1] := ConfigData.rec5_Pusher_Speed_1;
List_of_Recipes[5].Pusher.Speed[2] := ConfigData.rec5_Pusher_Speed_2;
List_of_Recipes[5].Pusher.Speed[3] := ConfigData.rec5_Pusher_Speed_3;
List_of_Recipes[5].Pusher.Speed[4] := ConfigData.rec5_Pusher_Speed_4;
List_of_Recipes[5].Pusher.Speed[5] := ConfigData.rec5_Pusher_Speed_5;
List_of_Recipes[5].Pusher.Speed[6] := ConfigData.rec5_Pusher_Speed_6;
List_of_Recipes[5].Pusher.distance[1] := ConfigData.rec5_Pusher_distance_1;
List_of_Recipes[5].Pusher.distance[2] := ConfigData.rec5_Pusher_distance_2;
List_of_Recipes[5].Pusher.distance[3] := ConfigData.rec5_Pusher_distance_3;
List_of_Recipes[5].Pusher.distance[4] := ConfigData.rec5_Pusher_distance_4;
List_of_Recipes[5].Pusher.distance[5] := ConfigData.rec5_Pusher_distance_5;
List_of_Recipes[5].Pusher.distance[6] := ConfigData.rec5_Pusher_distance_6;

List_of_Recipes[5].Compress.Initial_Distance := ConfigData.rec5_Compress_Initial_Distance;
List_of_Recipes[5].Compress.Initial_Speed := ConfigData.rec5_Compress_Initial_Speed;
List_of_Recipes[5].Compress.relax_Distance := ConfigData.rec5_Compress_Relax_Distance;
List_of_Recipes[5].Compress.retract_speed := ConfigData.rec5_Compress_retract_speed;

List_of_Recipes[5].Clamp.Release_Instance:=ConfigData.rec5_Clamp_Release_Instance;

List_of_Recipes[5].Other.Compress_Home_Offset:=ConfigData.rec5_Other_Compress_Home_Offset;
List_of_Recipes[5].Other.Shield_Home_Offset:=ConfigData.rec5_Other_Shield_Home_Offset;
List_of_Recipes[5].Other.Pusher_Home_Offset:=ConfigData.rec5_Other_Pusher_Home_Offset;

List_of_Recipes[5].Memory_Free:=LREAL_TO_BOOL(ConfigData.rec5_Memory_Free);	

//6
Rec_Name_1:=ConfigData.rec6_Name_1;								
Rec_Name_2:=ConfigData.rec6_Name_2;								
Rec_Name_3:=ConfigData.rec6_Name_3;								
Rec_Name_4:=ConfigData.rec6_Name_4;								
Rec_Name_5:=ConfigData.rec6_Name_5;
List_of_Recipes[6].Name:=Recipe_mem_name;

List_of_Recipes[6].Shield.Retract_Speed :=ConfigData.rec6_Shield_Retract_Speed;
List_of_Recipes[6].Shield.Speed[1] := ConfigData.rec6_Shield_Speed_1;
List_of_Recipes[6].Shield.Speed[2] := ConfigData.rec6_Shield_Speed_2;
List_of_Recipes[6].Shield.Speed[3] := ConfigData.rec6_Shield_Speed_3;
List_of_Recipes[6].Shield.Speed[4] := ConfigData.rec6_Shield_Speed_4;
List_of_Recipes[6].Shield.Speed[5] := ConfigData.rec6_Shield_Speed_5;
List_of_Recipes[6].Shield.Speed[6] := ConfigData.rec6_Shield_Speed_6;
List_of_Recipes[6].Shield.distance[1] := ConfigData.rec6_Shield_distance_1;
List_of_Recipes[6].Shield.distance[2] := ConfigData.rec6_Shield_distance_2;
List_of_Recipes[6].Shield.distance[3] := ConfigData.rec6_Shield_distance_3;
List_of_Recipes[6].Shield.distance[4] := ConfigData.rec6_Shield_distance_4;
List_of_Recipes[6].Shield.distance[5] := ConfigData.rec6_Shield_distance_5;
List_of_Recipes[6].Shield.distance[6] := ConfigData.rec6_Shield_distance_6;


List_of_Recipes[6].Pusher.Retract_Speed :=ConfigData.rec6_Pusher_Retract_Speed;
List_of_Recipes[6].Pusher.Speed[1] := ConfigData.rec6_Pusher_Speed_1;
List_of_Recipes[6].Pusher.Speed[2] := ConfigData.rec6_Pusher_Speed_2;
List_of_Recipes[6].Pusher.Speed[3] := ConfigData.rec6_Pusher_Speed_3;
List_of_Recipes[6].Pusher.Speed[4] := ConfigData.rec6_Pusher_Speed_4;
List_of_Recipes[6].Pusher.Speed[5] := ConfigData.rec6_Pusher_Speed_5;
List_of_Recipes[6].Pusher.Speed[6] := ConfigData.rec6_Pusher_Speed_6;
List_of_Recipes[6].Pusher.distance[1] := ConfigData.rec6_Pusher_distance_1;
List_of_Recipes[6].Pusher.distance[2] := ConfigData.rec6_Pusher_distance_2;
List_of_Recipes[6].Pusher.distance[3] := ConfigData.rec6_Pusher_distance_3;
List_of_Recipes[6].Pusher.distance[4] := ConfigData.rec6_Pusher_distance_4;
List_of_Recipes[6].Pusher.distance[5] := ConfigData.rec6_Pusher_distance_5;
List_of_Recipes[6].Pusher.distance[6] := ConfigData.rec6_Pusher_distance_6;

List_of_Recipes[6].Compress.Initial_Distance := ConfigData.rec6_Compress_Initial_Distance;
List_of_Recipes[6].Compress.Initial_Speed := ConfigData.rec6_Compress_Initial_Speed;
List_of_Recipes[6].Compress.relax_Distance := ConfigData.rec6_Compress_Relax_Distance;
List_of_Recipes[6].Compress.retract_speed := ConfigData.rec6_Compress_retract_speed;

List_of_Recipes[6].Clamp.Release_Instance:=ConfigData.rec6_Clamp_Release_Instance;

List_of_Recipes[6].Other.Compress_Home_Offset:=ConfigData.rec6_Other_Compress_Home_Offset;
List_of_Recipes[6].Other.Shield_Home_Offset:=ConfigData.rec6_Other_Shield_Home_Offset;
List_of_Recipes[6].Other.Pusher_Home_Offset:=ConfigData.rec6_Other_Pusher_Home_Offset;

List_of_Recipes[6].Memory_Free:=LREAL_TO_BOOL(ConfigData.rec6_Memory_Free);

//7
Rec_Name_1:=ConfigData.rec7_Name_1;								
Rec_Name_2:=ConfigData.rec7_Name_2;								
Rec_Name_3:=ConfigData.rec7_Name_3;								
Rec_Name_4:=ConfigData.rec7_Name_4;								
Rec_Name_5:=ConfigData.rec7_Name_5;
List_of_Recipes[7].Name:=Recipe_mem_name;

List_of_Recipes[7].Shield.Retract_Speed :=ConfigData.rec7_Shield_Retract_Speed;
List_of_Recipes[7].Shield.Speed[1] := ConfigData.rec7_Shield_Speed_1;
List_of_Recipes[7].Shield.Speed[2] := ConfigData.rec7_Shield_Speed_2;
List_of_Recipes[7].Shield.Speed[3] := ConfigData.rec7_Shield_Speed_3;
List_of_Recipes[7].Shield.Speed[4] := ConfigData.rec7_Shield_Speed_4;
List_of_Recipes[7].Shield.Speed[5] := ConfigData.rec7_Shield_Speed_5;
List_of_Recipes[7].Shield.Speed[6] := ConfigData.rec7_Shield_Speed_6;
List_of_Recipes[7].Shield.distance[1] := ConfigData.rec7_Shield_distance_1;
List_of_Recipes[7].Shield.distance[2] := ConfigData.rec7_Shield_distance_2;
List_of_Recipes[7].Shield.distance[3] := ConfigData.rec7_Shield_distance_3;
List_of_Recipes[7].Shield.distance[4] := ConfigData.rec7_Shield_distance_4;
List_of_Recipes[7].Shield.distance[5] := ConfigData.rec7_Shield_distance_5;
List_of_Recipes[7].Shield.distance[6] := ConfigData.rec7_Shield_distance_6;


List_of_Recipes[7].Pusher.Retract_Speed :=ConfigData.rec7_Pusher_Retract_Speed;
List_of_Recipes[7].Pusher.Speed[1] := ConfigData.rec7_Pusher_Speed_1;
List_of_Recipes[7].Pusher.Speed[2] := ConfigData.rec7_Pusher_Speed_2;
List_of_Recipes[7].Pusher.Speed[3] := ConfigData.rec7_Pusher_Speed_3;
List_of_Recipes[7].Pusher.Speed[4] := ConfigData.rec7_Pusher_Speed_4;
List_of_Recipes[7].Pusher.Speed[5] := ConfigData.rec7_Pusher_Speed_5;
List_of_Recipes[7].Pusher.Speed[6] := ConfigData.rec7_Pusher_Speed_6;
List_of_Recipes[7].Pusher.distance[1] := ConfigData.rec7_Pusher_distance_1;
List_of_Recipes[7].Pusher.distance[2] := ConfigData.rec7_Pusher_distance_2;
List_of_Recipes[7].Pusher.distance[3] := ConfigData.rec7_Pusher_distance_3;
List_of_Recipes[7].Pusher.distance[4] := ConfigData.rec7_Pusher_distance_4;
List_of_Recipes[7].Pusher.distance[5] := ConfigData.rec7_Pusher_distance_5;
List_of_Recipes[7].Pusher.distance[6] := ConfigData.rec7_Pusher_distance_6;

List_of_Recipes[7].Compress.Initial_Distance := ConfigData.rec7_Compress_Initial_Distance;
List_of_Recipes[7].Compress.Initial_Speed := ConfigData.rec7_Compress_Initial_Speed;
List_of_Recipes[7].Compress.relax_Distance := ConfigData.rec7_Compress_Relax_Distance;
List_of_Recipes[7].Compress.retract_speed := ConfigData.rec7_Compress_retract_speed;

List_of_Recipes[7].Clamp.Release_Instance:=ConfigData.rec7_Clamp_Release_Instance;

List_of_Recipes[7].Other.Compress_Home_Offset:=ConfigData.rec7_Other_Compress_Home_Offset;
List_of_Recipes[7].Other.Shield_Home_Offset:=ConfigData.rec7_Other_Shield_Home_Offset;
List_of_Recipes[7].Other.Pusher_Home_Offset:=ConfigData.rec7_Other_Pusher_Home_Offset;

List_of_Recipes[7].Memory_Free:=LREAL_TO_BOOL(ConfigData.rec7_Memory_Free);	
	
//8
Rec_Name_1:=ConfigData.rec8_Name_1;								
Rec_Name_2:=ConfigData.rec8_Name_2;								
Rec_Name_3:=ConfigData.rec8_Name_3;								
Rec_Name_4:=ConfigData.rec8_Name_4;								
Rec_Name_5:=ConfigData.rec8_Name_5;
List_of_Recipes[8].Name:=Recipe_mem_name;

List_of_Recipes[8].Shield.Retract_Speed :=ConfigData.rec8_Shield_Retract_Speed;
List_of_Recipes[8].Shield.Speed[1] := ConfigData.rec8_Shield_Speed_1;
List_of_Recipes[8].Shield.Speed[2] := ConfigData.rec8_Shield_Speed_2;
List_of_Recipes[8].Shield.Speed[3] := ConfigData.rec8_Shield_Speed_3;
List_of_Recipes[8].Shield.Speed[4] := ConfigData.rec8_Shield_Speed_4;
List_of_Recipes[8].Shield.Speed[5] := ConfigData.rec8_Shield_Speed_5;
List_of_Recipes[8].Shield.Speed[6] := ConfigData.rec8_Shield_Speed_6;
List_of_Recipes[8].Shield.distance[1] := ConfigData.rec8_Shield_distance_1;
List_of_Recipes[8].Shield.distance[2] := ConfigData.rec8_Shield_distance_2;
List_of_Recipes[8].Shield.distance[3] := ConfigData.rec8_Shield_distance_3;
List_of_Recipes[8].Shield.distance[4] := ConfigData.rec8_Shield_distance_4;
List_of_Recipes[8].Shield.distance[5] := ConfigData.rec8_Shield_distance_5;
List_of_Recipes[8].Shield.distance[6] := ConfigData.rec8_Shield_distance_6;


List_of_Recipes[8].Pusher.Retract_Speed :=ConfigData.rec8_Pusher_Retract_Speed;
List_of_Recipes[8].Pusher.Speed[1] := ConfigData.rec8_Pusher_Speed_1;
List_of_Recipes[8].Pusher.Speed[2] := ConfigData.rec8_Pusher_Speed_2;
List_of_Recipes[8].Pusher.Speed[3] := ConfigData.rec8_Pusher_Speed_3;
List_of_Recipes[8].Pusher.Speed[4] := ConfigData.rec8_Pusher_Speed_4;
List_of_Recipes[8].Pusher.Speed[5] := ConfigData.rec8_Pusher_Speed_5;
List_of_Recipes[8].Pusher.Speed[6] := ConfigData.rec8_Pusher_Speed_6;
List_of_Recipes[8].Pusher.distance[1] := ConfigData.rec8_Pusher_distance_1;
List_of_Recipes[8].Pusher.distance[2] := ConfigData.rec8_Pusher_distance_2;
List_of_Recipes[8].Pusher.distance[3] := ConfigData.rec8_Pusher_distance_3;
List_of_Recipes[8].Pusher.distance[4] := ConfigData.rec8_Pusher_distance_4;
List_of_Recipes[8].Pusher.distance[5] := ConfigData.rec8_Pusher_distance_5;
List_of_Recipes[8].Pusher.distance[6] := ConfigData.rec8_Pusher_distance_6;

List_of_Recipes[8].Compress.Initial_Distance := ConfigData.rec8_Compress_Initial_Distance;
List_of_Recipes[8].Compress.Initial_Speed := ConfigData.rec8_Compress_Initial_Speed;
List_of_Recipes[8].Compress.relax_Distance := ConfigData.rec8_Compress_Relax_Distance;
List_of_Recipes[8].Compress.retract_speed := ConfigData.rec8_Compress_retract_speed;

List_of_Recipes[8].Clamp.Release_Instance:=ConfigData.rec8_Clamp_Release_Instance;

List_of_Recipes[8].Other.Compress_Home_Offset:=ConfigData.rec8_Other_Compress_Home_Offset;
List_of_Recipes[8].Other.Shield_Home_Offset:=ConfigData.rec8_Other_Shield_Home_Offset;
List_of_Recipes[8].Other.Pusher_Home_Offset:=ConfigData.rec8_Other_Pusher_Home_Offset;

List_of_Recipes[8].Memory_Free:=LREAL_TO_BOOL(ConfigData.rec8_Memory_Free);	

//9
Rec_Name_1:=ConfigData.rec9_Name_1;								
Rec_Name_2:=ConfigData.rec9_Name_2;								
Rec_Name_3:=ConfigData.rec9_Name_3;								
Rec_Name_4:=ConfigData.rec9_Name_4;								
Rec_Name_5:=ConfigData.rec9_Name_5;
List_of_Recipes[9].Name:=Recipe_mem_name;

List_of_Recipes[9].Shield.Retract_Speed :=ConfigData.rec9_Shield_Retract_Speed;
List_of_Recipes[9].Shield.Speed[1] := ConfigData.rec9_Shield_Speed_1;
List_of_Recipes[9].Shield.Speed[2] := ConfigData.rec9_Shield_Speed_2;
List_of_Recipes[9].Shield.Speed[3] := ConfigData.rec9_Shield_Speed_3;
List_of_Recipes[9].Shield.Speed[4] := ConfigData.rec9_Shield_Speed_4;
List_of_Recipes[9].Shield.Speed[5] := ConfigData.rec9_Shield_Speed_5;
List_of_Recipes[9].Shield.Speed[6] := ConfigData.rec9_Shield_Speed_6;
List_of_Recipes[9].Shield.distance[1] := ConfigData.rec9_Shield_distance_1;
List_of_Recipes[9].Shield.distance[2] := ConfigData.rec9_Shield_distance_2;
List_of_Recipes[9].Shield.distance[3] := ConfigData.rec9_Shield_distance_3;
List_of_Recipes[9].Shield.distance[4] := ConfigData.rec9_Shield_distance_4;
List_of_Recipes[9].Shield.distance[5] := ConfigData.rec9_Shield_distance_5;
List_of_Recipes[9].Shield.distance[6] := ConfigData.rec9_Shield_distance_6;


List_of_Recipes[9].Pusher.Retract_Speed :=ConfigData.rec9_Pusher_Retract_Speed;
List_of_Recipes[9].Pusher.Speed[1] := ConfigData.rec9_Pusher_Speed_1;
List_of_Recipes[9].Pusher.Speed[2] := ConfigData.rec9_Pusher_Speed_2;
List_of_Recipes[9].Pusher.Speed[3] := ConfigData.rec9_Pusher_Speed_3;
List_of_Recipes[9].Pusher.Speed[4] := ConfigData.rec9_Pusher_Speed_4;
List_of_Recipes[9].Pusher.Speed[5] := ConfigData.rec9_Pusher_Speed_5;
List_of_Recipes[9].Pusher.Speed[6] := ConfigData.rec9_Pusher_Speed_6;
List_of_Recipes[9].Pusher.distance[1] := ConfigData.rec9_Pusher_distance_1;
List_of_Recipes[9].Pusher.distance[2] := ConfigData.rec9_Pusher_distance_2;
List_of_Recipes[9].Pusher.distance[3] := ConfigData.rec9_Pusher_distance_3;
List_of_Recipes[9].Pusher.distance[4] := ConfigData.rec9_Pusher_distance_4;
List_of_Recipes[9].Pusher.distance[5] := ConfigData.rec9_Pusher_distance_5;
List_of_Recipes[9].Pusher.distance[6] := ConfigData.rec9_Pusher_distance_6;

List_of_Recipes[9].Compress.Initial_Distance := ConfigData.rec9_Compress_Initial_Distance;
List_of_Recipes[9].Compress.Initial_Speed := ConfigData.rec9_Compress_Initial_Speed;
List_of_Recipes[9].Compress.relax_Distance := ConfigData.rec9_Compress_Relax_Distance;
List_of_Recipes[9].Compress.retract_speed := ConfigData.rec9_Compress_retract_speed;

List_of_Recipes[9].Clamp.Release_Instance:=ConfigData.rec9_Clamp_Release_Instance;

List_of_Recipes[9].Other.Compress_Home_Offset:=ConfigData.rec9_Other_Compress_Home_Offset;
List_of_Recipes[9].Other.Shield_Home_Offset:=ConfigData.rec9_Other_Shield_Home_Offset;
List_of_Recipes[9].Other.Pusher_Home_Offset:=ConfigData.rec9_Other_Pusher_Home_Offset;

List_of_Recipes[9].Memory_Free:=LREAL_TO_BOOL(ConfigData.rec9_Memory_Free);	

//10
Rec_Name_1:=ConfigData.rec10_Name_1;								
Rec_Name_2:=ConfigData.rec10_Name_2;								
Rec_Name_3:=ConfigData.rec10_Name_3;								
Rec_Name_4:=ConfigData.rec10_Name_4;								
Rec_Name_5:=ConfigData.rec10_Name_5;
List_of_Recipes[10].Name:=Recipe_mem_name;

List_of_Recipes[10].Shield.Retract_Speed :=ConfigData.rec10_Shield_Retract_Speed;
List_of_Recipes[10].Shield.Speed[1] := ConfigData.rec10_Shield_Speed_1;
List_of_Recipes[10].Shield.Speed[2] := ConfigData.rec10_Shield_Speed_2;
List_of_Recipes[10].Shield.Speed[3] := ConfigData.rec10_Shield_Speed_3;
List_of_Recipes[10].Shield.Speed[4] := ConfigData.rec10_Shield_Speed_4;
List_of_Recipes[10].Shield.Speed[5] := ConfigData.rec10_Shield_Speed_5;
List_of_Recipes[10].Shield.Speed[6] := ConfigData.rec10_Shield_Speed_6;
List_of_Recipes[10].Shield.distance[1] := ConfigData.rec10_Shield_distance_1;
List_of_Recipes[10].Shield.distance[2] := ConfigData.rec10_Shield_distance_2;
List_of_Recipes[10].Shield.distance[3] := ConfigData.rec10_Shield_distance_3;
List_of_Recipes[10].Shield.distance[4] := ConfigData.rec10_Shield_distance_4;
List_of_Recipes[10].Shield.distance[5] := ConfigData.rec10_Shield_distance_5;
List_of_Recipes[10].Shield.distance[6] := ConfigData.rec10_Shield_distance_6;


List_of_Recipes[10].Pusher.Retract_Speed :=ConfigData.rec10_Pusher_Retract_Speed;
List_of_Recipes[10].Pusher.Speed[1] := ConfigData.rec10_Pusher_Speed_1;
List_of_Recipes[10].Pusher.Speed[2] := ConfigData.rec10_Pusher_Speed_2;
List_of_Recipes[10].Pusher.Speed[3] := ConfigData.rec10_Pusher_Speed_3;
List_of_Recipes[10].Pusher.Speed[4] := ConfigData.rec10_Pusher_Speed_4;
List_of_Recipes[10].Pusher.Speed[5] := ConfigData.rec10_Pusher_Speed_5;
List_of_Recipes[10].Pusher.Speed[6] := ConfigData.rec10_Pusher_Speed_6;
List_of_Recipes[10].Pusher.distance[1] := ConfigData.rec10_Pusher_distance_1;
List_of_Recipes[10].Pusher.distance[2] := ConfigData.rec10_Pusher_distance_2;
List_of_Recipes[10].Pusher.distance[3] := ConfigData.rec10_Pusher_distance_3;
List_of_Recipes[10].Pusher.distance[4] := ConfigData.rec10_Pusher_distance_4;
List_of_Recipes[10].Pusher.distance[5] := ConfigData.rec10_Pusher_distance_5;
List_of_Recipes[10].Pusher.distance[6] := ConfigData.rec10_Pusher_distance_6;

List_of_Recipes[10].Compress.Initial_Distance := ConfigData.rec10_Compress_Initial_Distance;
List_of_Recipes[10].Compress.Initial_Speed := ConfigData.rec10_Compress_Initial_Speed;
List_of_Recipes[10].Compress.relax_Distance := ConfigData.rec10_Compress_Relax_Distance;
List_of_Recipes[10].Compress.retract_speed := ConfigData.rec10_Compress_retract_speed;

List_of_Recipes[10].Clamp.Release_Instance:=ConfigData.rec10_Clamp_Release_Instance;

List_of_Recipes[10].Other.Compress_Home_Offset:=ConfigData.rec10_Other_Compress_Home_Offset;
List_of_Recipes[10].Other.Shield_Home_Offset:=ConfigData.rec10_Other_Shield_Home_Offset;
List_of_Recipes[10].Other.Pusher_Home_Offset:=ConfigData.rec10_Other_Pusher_Home_Offset;

List_of_Recipes[10].Memory_Free:=LREAL_TO_BOOL(ConfigData.rec10_Memory_Free);
END_METHOD

METHOD CopyGlobalRecipiesToConfig : BOOL
VAR_INPUT

END_VAR

VAR
	List_of_RRecipes: INT;
END_VAR



ConfigData.con_max_limit_Compress:=limits_save.max_limit_Compress;
ConfigData.con_max_limit_Pusher:=Limits_save.max_limit_Pusher;
ConfigData.con_max_limit_Shield:=Limits_save.max_limit_Shield;
ConfigData.con_max_pusher_shield_diff:=Limits_save.max_pusher_shield_diff;
ConfigData.con_max_torque:=Limits_save.max_torque;	

//1

Recipe_mem_name := List_of_Recipes[1].Name;

ConfigData.rec1_Name_1:=Rec_Name_1;								
ConfigData.rec1_Name_2:=Rec_Name_2;								
ConfigData.rec1_Name_3:=Rec_Name_3;								
ConfigData.rec1_Name_4:=Rec_Name_4;								
ConfigData.rec1_Name_5:=Rec_Name_5;

ConfigData.rec1_Shield_Retract_Speed := List_of_Recipes[1].Shield.Retract_Speed;
ConfigData.rec1_Shield_Speed_1 := List_of_Recipes[1].Shield.Speed[1];
ConfigData.rec1_Shield_Speed_2 := List_of_Recipes[1].Shield.Speed[2];
ConfigData.rec1_Shield_Speed_3 := List_of_Recipes[1].Shield.Speed[3];
ConfigData.rec1_Shield_Speed_4 := List_of_Recipes[1].Shield.Speed[4];
ConfigData.rec1_Shield_Speed_5 := List_of_Recipes[1].Shield.Speed[5];
ConfigData.rec1_Shield_Speed_6 := List_of_Recipes[1].Shield.Speed[6];
ConfigData.rec1_Shield_distance_1 := List_of_Recipes[1].Shield.distance[1];
ConfigData.rec1_Shield_distance_2 := List_of_Recipes[1].Shield.distance[2];
ConfigData.rec1_Shield_distance_3 := List_of_Recipes[1].Shield.distance[3];
ConfigData.rec1_Shield_distance_4 := List_of_Recipes[1].Shield.distance[4];
ConfigData.rec1_Shield_distance_5 := List_of_Recipes[1].Shield.distance[5];
ConfigData.rec1_Shield_distance_6 := List_of_Recipes[1].Shield.distance[6];


ConfigData.rec1_Pusher_Retract_Speed := List_of_Recipes[1].Pusher.Retract_Speed;
ConfigData.rec1_Pusher_Speed_1 := List_of_Recipes[1].Pusher.Speed[1];
ConfigData.rec1_Pusher_Speed_2 := List_of_Recipes[1].Pusher.Speed[2];
ConfigData.rec1_Pusher_Speed_3 := List_of_Recipes[1].Pusher.Speed[3];
ConfigData.rec1_Pusher_Speed_4 := List_of_Recipes[1].Pusher.Speed[4];
ConfigData.rec1_Pusher_Speed_5 := List_of_Recipes[1].Pusher.Speed[5];
ConfigData.rec1_Pusher_Speed_6 := List_of_Recipes[1].Pusher.Speed[6];
ConfigData.rec1_Pusher_distance_1 := List_of_Recipes[1].Pusher.distance[1];
ConfigData.rec1_Pusher_distance_2 := List_of_Recipes[1].Pusher.distance[2];
ConfigData.rec1_Pusher_distance_3 := List_of_Recipes[1].Pusher.distance[3];
ConfigData.rec1_Pusher_distance_4 := List_of_Recipes[1].Pusher.distance[4];
ConfigData.rec1_Pusher_distance_5 := List_of_Recipes[1].Pusher.distance[5];
ConfigData.rec1_Pusher_distance_6 := List_of_Recipes[1].Pusher.distance[6];

ConfigData.rec1_Compress_Initial_Distance:= List_of_Recipes[1].Compress.Initial_Distance;
ConfigData.rec1_Compress_Initial_Speed:= List_of_Recipes[1].Compress.Initial_Speed;
ConfigData.rec1_Compress_Relax_Distance:=List_of_Recipes[1].Compress.Relax_Distance;
ConfigData.rec1_Compress_Retract_Speed:=List_of_Recipes[1].Compress.Retract_Speed;

ConfigData.rec1_Clamp_Release_Instance:=List_of_Recipes[1].Clamp.Release_Instance;

ConfigData.rec1_Other_Compress_Home_Offset:=List_of_Recipes[1].Other.Compress_Home_Offset;
ConfigData.rec1_Other_Shield_Home_Offset:=List_of_Recipes[1].Other.Shield_Home_Offset;
ConfigData.rec1_Other_Pusher_Home_Offset:=List_of_Recipes[1].Other.Pusher_Home_Offset;

ConfigData.rec1_Memory_Free:=BOOL_TO_LREAL(List_of_Recipes[1].Memory_Free);


//2


Recipe_mem_name := List_of_Recipes[2].Name;

ConfigData.rec2_Name_1:=Rec_Name_1;								
ConfigData.rec2_Name_2:=Rec_Name_2;								
ConfigData.rec2_Name_3:=Rec_Name_3;								
ConfigData.rec2_Name_4:=Rec_Name_4;								
ConfigData.rec2_Name_5:=Rec_Name_5;

ConfigData.rec2_Shield_Retract_Speed := List_of_Recipes[2].Shield.Retract_Speed;
ConfigData.rec2_Shield_Speed_1 := List_of_Recipes[2].Shield.Speed[1];
ConfigData.rec2_Shield_Speed_2 := List_of_Recipes[2].Shield.Speed[2];
ConfigData.rec2_Shield_Speed_3 := List_of_Recipes[2].Shield.Speed[3];
ConfigData.rec2_Shield_Speed_4 := List_of_Recipes[2].Shield.Speed[4];
ConfigData.rec2_Shield_Speed_5 := List_of_Recipes[2].Shield.Speed[5];
ConfigData.rec2_Shield_Speed_6 := List_of_Recipes[2].Shield.Speed[6];
ConfigData.rec2_Shield_distance_1 := List_of_Recipes[2].Shield.distance[1];
ConfigData.rec2_Shield_distance_2 := List_of_Recipes[2].Shield.distance[2];
ConfigData.rec2_Shield_distance_3 := List_of_Recipes[2].Shield.distance[3];
ConfigData.rec2_Shield_distance_4 := List_of_Recipes[2].Shield.distance[4];
ConfigData.rec2_Shield_distance_5 := List_of_Recipes[2].Shield.distance[5];
ConfigData.rec2_Shield_distance_6 := List_of_Recipes[2].Shield.distance[6];


ConfigData.rec2_Pusher_Retract_Speed := List_of_Recipes[2].Pusher.Retract_Speed;
ConfigData.rec2_Pusher_Speed_1 := List_of_Recipes[2].Pusher.Speed[1];
ConfigData.rec2_Pusher_Speed_2 := List_of_Recipes[2].Pusher.Speed[2];
ConfigData.rec2_Pusher_Speed_3 := List_of_Recipes[2].Pusher.Speed[3];
ConfigData.rec2_Pusher_Speed_4 := List_of_Recipes[2].Pusher.Speed[4];
ConfigData.rec2_Pusher_Speed_5 := List_of_Recipes[2].Pusher.Speed[5];
ConfigData.rec2_Pusher_Speed_6 := List_of_Recipes[2].Pusher.Speed[6];
ConfigData.rec2_Pusher_distance_1 := List_of_Recipes[2].Pusher.distance[1];
ConfigData.rec2_Pusher_distance_2 := List_of_Recipes[2].Pusher.distance[2];
ConfigData.rec2_Pusher_distance_3 := List_of_Recipes[2].Pusher.distance[3];
ConfigData.rec2_Pusher_distance_4 := List_of_Recipes[2].Pusher.distance[4];
ConfigData.rec2_Pusher_distance_5 := List_of_Recipes[2].Pusher.distance[5];
ConfigData.rec2_Pusher_distance_6 := List_of_Recipes[2].Pusher.distance[6];

ConfigData.rec2_Compress_Initial_Distance:= List_of_Recipes[2].Compress.Initial_Distance;
ConfigData.rec2_Compress_Initial_Speed:= List_of_Recipes[2].Compress.Initial_Speed;
ConfigData.rec2_Compress_Relax_Distance:=List_of_Recipes[2].Compress.Relax_Distance;
ConfigData.rec2_Compress_Retract_Speed:=List_of_Recipes[2].Compress.Retract_Speed;

ConfigData.rec2_Clamp_Release_Instance:=List_of_Recipes[2].Clamp.Release_Instance;

ConfigData.rec2_Other_Compress_Home_Offset:=List_of_Recipes[2].Other.Compress_Home_Offset;
ConfigData.rec2_Other_Shield_Home_Offset:=List_of_Recipes[2].Other.Shield_Home_Offset;
ConfigData.rec2_Other_Pusher_Home_Offset:=List_of_Recipes[2].Other.Pusher_Home_Offset;

ConfigData.rec2_Memory_Free:=BOOL_TO_LREAL(List_of_Recipes[2].Memory_Free);

//3


Recipe_mem_name := List_of_Recipes[3].Name;

ConfigData.rec3_Name_1:=Rec_Name_1;								
ConfigData.rec3_Name_2:=Rec_Name_2;								
ConfigData.rec3_Name_3:=Rec_Name_3;								
ConfigData.rec3_Name_4:=Rec_Name_4;								
ConfigData.rec3_Name_5:=Rec_Name_5;

ConfigData.rec3_Shield_Retract_Speed := List_of_Recipes[3].Shield.Retract_Speed;
ConfigData.rec3_Shield_Speed_1 := List_of_Recipes[3].Shield.Speed[1];
ConfigData.rec3_Shield_Speed_2 := List_of_Recipes[3].Shield.Speed[2];
ConfigData.rec3_Shield_Speed_3 := List_of_Recipes[3].Shield.Speed[3];
ConfigData.rec3_Shield_Speed_4 := List_of_Recipes[3].Shield.Speed[4];
ConfigData.rec3_Shield_Speed_5 := List_of_Recipes[3].Shield.Speed[5];
ConfigData.rec3_Shield_Speed_6 := List_of_Recipes[3].Shield.Speed[6];
ConfigData.rec3_Shield_distance_1 := List_of_Recipes[3].Shield.distance[1];
ConfigData.rec3_Shield_distance_2 := List_of_Recipes[3].Shield.distance[2];
ConfigData.rec3_Shield_distance_3 := List_of_Recipes[3].Shield.distance[3];
ConfigData.rec3_Shield_distance_4 := List_of_Recipes[3].Shield.distance[4];
ConfigData.rec3_Shield_distance_5 := List_of_Recipes[3].Shield.distance[5];
ConfigData.rec3_Shield_distance_6 := List_of_Recipes[3].Shield.distance[6];


ConfigData.rec3_Pusher_Retract_Speed := List_of_Recipes[3].Pusher.Retract_Speed;
ConfigData.rec3_Pusher_Speed_1 := List_of_Recipes[3].Pusher.Speed[1];
ConfigData.rec3_Pusher_Speed_2 := List_of_Recipes[3].Pusher.Speed[2];
ConfigData.rec3_Pusher_Speed_3 := List_of_Recipes[3].Pusher.Speed[3];
ConfigData.rec3_Pusher_Speed_4 := List_of_Recipes[3].Pusher.Speed[4];
ConfigData.rec3_Pusher_Speed_5 := List_of_Recipes[3].Pusher.Speed[5];
ConfigData.rec3_Pusher_Speed_6 := List_of_Recipes[3].Pusher.Speed[6];
ConfigData.rec3_Pusher_distance_1 := List_of_Recipes[3].Pusher.distance[1];
ConfigData.rec3_Pusher_distance_2 := List_of_Recipes[3].Pusher.distance[2];
ConfigData.rec3_Pusher_distance_3 := List_of_Recipes[3].Pusher.distance[3];
ConfigData.rec3_Pusher_distance_4 := List_of_Recipes[3].Pusher.distance[4];
ConfigData.rec3_Pusher_distance_5 := List_of_Recipes[3].Pusher.distance[5];
ConfigData.rec3_Pusher_distance_6 := List_of_Recipes[3].Pusher.distance[6];

ConfigData.rec3_Compress_Initial_Distance:= List_of_Recipes[3].Compress.Initial_Distance;
ConfigData.rec3_Compress_Initial_Speed:= List_of_Recipes[3].Compress.Initial_Speed;
ConfigData.rec3_Compress_Relax_Distance:=List_of_Recipes[3].Compress.Relax_Distance;
ConfigData.rec3_Compress_Retract_Speed:=List_of_Recipes[3].Compress.Retract_Speed;

ConfigData.rec3_Clamp_Release_Instance:=List_of_Recipes[3].Clamp.Release_Instance;

ConfigData.rec3_Other_Compress_Home_Offset:=List_of_Recipes[3].Other.Compress_Home_Offset;
ConfigData.rec3_Other_Shield_Home_Offset:=List_of_Recipes[3].Other.Shield_Home_Offset;
ConfigData.rec3_Other_Pusher_Home_Offset:=List_of_Recipes[3].Other.Pusher_Home_Offset;

ConfigData.rec3_Memory_Free:=BOOL_TO_LREAL(List_of_Recipes[3].Memory_Free);

//4


Recipe_mem_name := List_of_Recipes[4].Name;

ConfigData.rec4_Name_1:=Rec_Name_1;								
ConfigData.rec4_Name_2:=Rec_Name_2;								
ConfigData.rec4_Name_3:=Rec_Name_3;								
ConfigData.rec4_Name_4:=Rec_Name_4;								
ConfigData.rec4_Name_5:=Rec_Name_5;

ConfigData.rec4_Shield_Retract_Speed := List_of_Recipes[4].Shield.Retract_Speed;
ConfigData.rec4_Shield_Speed_1 := List_of_Recipes[4].Shield.Speed[1];
ConfigData.rec4_Shield_Speed_2 := List_of_Recipes[4].Shield.Speed[2];
ConfigData.rec4_Shield_Speed_3 := List_of_Recipes[4].Shield.Speed[3];
ConfigData.rec4_Shield_Speed_4 := List_of_Recipes[4].Shield.Speed[4];
ConfigData.rec4_Shield_Speed_5 := List_of_Recipes[4].Shield.Speed[5];
ConfigData.rec4_Shield_Speed_6 := List_of_Recipes[4].Shield.Speed[6];
ConfigData.rec4_Shield_distance_1 := List_of_Recipes[4].Shield.distance[1];
ConfigData.rec4_Shield_distance_2 := List_of_Recipes[4].Shield.distance[2];
ConfigData.rec4_Shield_distance_3 := List_of_Recipes[4].Shield.distance[3];
ConfigData.rec4_Shield_distance_4 := List_of_Recipes[4].Shield.distance[4];
ConfigData.rec4_Shield_distance_5 := List_of_Recipes[4].Shield.distance[5];
ConfigData.rec4_Shield_distance_6 := List_of_Recipes[4].Shield.distance[6];


ConfigData.rec4_Pusher_Retract_Speed := List_of_Recipes[4].Pusher.Retract_Speed;
ConfigData.rec4_Pusher_Speed_1 := List_of_Recipes[4].Pusher.Speed[1];
ConfigData.rec4_Pusher_Speed_2 := List_of_Recipes[4].Pusher.Speed[2];
ConfigData.rec4_Pusher_Speed_3 := List_of_Recipes[4].Pusher.Speed[3];
ConfigData.rec4_Pusher_Speed_4 := List_of_Recipes[4].Pusher.Speed[4];
ConfigData.rec4_Pusher_Speed_5 := List_of_Recipes[4].Pusher.Speed[5];
ConfigData.rec4_Pusher_Speed_6 := List_of_Recipes[4].Pusher.Speed[6];
ConfigData.rec4_Pusher_distance_1 := List_of_Recipes[4].Pusher.distance[1];
ConfigData.rec4_Pusher_distance_2 := List_of_Recipes[4].Pusher.distance[2];
ConfigData.rec4_Pusher_distance_3 := List_of_Recipes[4].Pusher.distance[3];
ConfigData.rec4_Pusher_distance_4 := List_of_Recipes[4].Pusher.distance[4];
ConfigData.rec4_Pusher_distance_5 := List_of_Recipes[4].Pusher.distance[5];
ConfigData.rec4_Pusher_distance_6 := List_of_Recipes[4].Pusher.distance[6];

ConfigData.rec4_Compress_Initial_Distance:= List_of_Recipes[4].Compress.Initial_Distance;
ConfigData.rec4_Compress_Initial_Speed:= List_of_Recipes[4].Compress.Initial_Speed;
ConfigData.rec4_Compress_Relax_Distance:=List_of_Recipes[4].Compress.Relax_Distance;
ConfigData.rec4_Compress_Retract_Speed:=List_of_Recipes[4].Compress.Retract_Speed;

ConfigData.rec4_Clamp_Release_Instance:=List_of_Recipes[4].Clamp.Release_Instance;

ConfigData.rec4_Other_Compress_Home_Offset:=List_of_Recipes[4].Other.Compress_Home_Offset;
ConfigData.rec4_Other_Shield_Home_Offset:=List_of_Recipes[4].Other.Shield_Home_Offset;
ConfigData.rec4_Other_Pusher_Home_Offset:=List_of_Recipes[4].Other.Pusher_Home_Offset;

ConfigData.rec4_Memory_Free:=BOOL_TO_LREAL(List_of_Recipes[4].Memory_Free);

//5


Recipe_mem_name := List_of_Recipes[5].Name;

ConfigData.rec5_Name_1:=Rec_Name_1;								
ConfigData.rec5_Name_2:=Rec_Name_2;								
ConfigData.rec5_Name_3:=Rec_Name_3;								
ConfigData.rec5_Name_4:=Rec_Name_4;								
ConfigData.rec5_Name_5:=Rec_Name_5;

ConfigData.rec5_Shield_Retract_Speed := List_of_Recipes[5].Shield.Retract_Speed;
ConfigData.rec5_Shield_Speed_1 := List_of_Recipes[5].Shield.Speed[1];
ConfigData.rec5_Shield_Speed_2 := List_of_Recipes[5].Shield.Speed[2];
ConfigData.rec5_Shield_Speed_3 := List_of_Recipes[5].Shield.Speed[3];
ConfigData.rec5_Shield_Speed_4 := List_of_Recipes[5].Shield.Speed[4];
ConfigData.rec5_Shield_Speed_5 := List_of_Recipes[5].Shield.Speed[5];
ConfigData.rec5_Shield_Speed_6 := List_of_Recipes[5].Shield.Speed[6];
ConfigData.rec5_Shield_distance_1 := List_of_Recipes[5].Shield.distance[1];
ConfigData.rec5_Shield_distance_2 := List_of_Recipes[5].Shield.distance[2];
ConfigData.rec5_Shield_distance_3 := List_of_Recipes[5].Shield.distance[3];
ConfigData.rec5_Shield_distance_4 := List_of_Recipes[5].Shield.distance[4];
ConfigData.rec5_Shield_distance_5 := List_of_Recipes[5].Shield.distance[5];
ConfigData.rec5_Shield_distance_6 := List_of_Recipes[5].Shield.distance[6];


ConfigData.rec5_Pusher_Retract_Speed := List_of_Recipes[5].Pusher.Retract_Speed;
ConfigData.rec5_Pusher_Speed_1 := List_of_Recipes[5].Pusher.Speed[1];
ConfigData.rec5_Pusher_Speed_2 := List_of_Recipes[5].Pusher.Speed[2];
ConfigData.rec5_Pusher_Speed_3 := List_of_Recipes[5].Pusher.Speed[3];
ConfigData.rec5_Pusher_Speed_4 := List_of_Recipes[5].Pusher.Speed[4];
ConfigData.rec5_Pusher_Speed_5 := List_of_Recipes[5].Pusher.Speed[5];
ConfigData.rec5_Pusher_Speed_6 := List_of_Recipes[5].Pusher.Speed[6];
ConfigData.rec5_Pusher_distance_1 := List_of_Recipes[5].Pusher.distance[1];
ConfigData.rec5_Pusher_distance_2 := List_of_Recipes[5].Pusher.distance[2];
ConfigData.rec5_Pusher_distance_3 := List_of_Recipes[5].Pusher.distance[3];
ConfigData.rec5_Pusher_distance_4 := List_of_Recipes[5].Pusher.distance[4];
ConfigData.rec5_Pusher_distance_5 := List_of_Recipes[5].Pusher.distance[5];
ConfigData.rec5_Pusher_distance_6 := List_of_Recipes[5].Pusher.distance[6];

ConfigData.rec5_Compress_Initial_Distance:= List_of_Recipes[5].Compress.Initial_Distance;
ConfigData.rec5_Compress_Initial_Speed:= List_of_Recipes[5].Compress.Initial_Speed;
ConfigData.rec5_Compress_Relax_Distance:=List_of_Recipes[5].Compress.Relax_Distance;
ConfigData.rec5_Compress_Retract_Speed:=List_of_Recipes[5].Compress.Retract_Speed;

ConfigData.rec5_Clamp_Release_Instance:=List_of_Recipes[5].Clamp.Release_Instance;

ConfigData.rec5_Other_Compress_Home_Offset:=List_of_Recipes[5].Other.Compress_Home_Offset;
ConfigData.rec5_Other_Shield_Home_Offset:=List_of_Recipes[5].Other.Shield_Home_Offset;
ConfigData.rec5_Other_Pusher_Home_Offset:=List_of_Recipes[5].Other.Pusher_Home_Offset;

ConfigData.rec5_Memory_Free:=BOOL_TO_LREAL(List_of_Recipes[5].Memory_Free);

//6


Recipe_mem_name := List_of_Recipes[6].Name;

ConfigData.rec6_Name_1:=Rec_Name_1;								
ConfigData.rec6_Name_2:=Rec_Name_2;								
ConfigData.rec6_Name_3:=Rec_Name_3;								
ConfigData.rec6_Name_4:=Rec_Name_4;								
ConfigData.rec6_Name_5:=Rec_Name_5;

ConfigData.rec6_Shield_Retract_Speed := List_of_Recipes[6].Shield.Retract_Speed;
ConfigData.rec6_Shield_Speed_1 := List_of_Recipes[6].Shield.Speed[1];
ConfigData.rec6_Shield_Speed_2 := List_of_Recipes[6].Shield.Speed[2];
ConfigData.rec6_Shield_Speed_3 := List_of_Recipes[6].Shield.Speed[3];
ConfigData.rec6_Shield_Speed_4 := List_of_Recipes[6].Shield.Speed[4];
ConfigData.rec6_Shield_Speed_5 := List_of_Recipes[6].Shield.Speed[5];
ConfigData.rec6_Shield_Speed_6 := List_of_Recipes[6].Shield.Speed[6];
ConfigData.rec6_Shield_distance_1 := List_of_Recipes[6].Shield.distance[1];
ConfigData.rec6_Shield_distance_2 := List_of_Recipes[6].Shield.distance[2];
ConfigData.rec6_Shield_distance_3 := List_of_Recipes[6].Shield.distance[3];
ConfigData.rec6_Shield_distance_4 := List_of_Recipes[6].Shield.distance[4];
ConfigData.rec6_Shield_distance_5 := List_of_Recipes[6].Shield.distance[5];
ConfigData.rec6_Shield_distance_6 := List_of_Recipes[6].Shield.distance[6];


ConfigData.rec6_Pusher_Retract_Speed := List_of_Recipes[6].Pusher.Retract_Speed;
ConfigData.rec6_Pusher_Speed_1 := List_of_Recipes[6].Pusher.Speed[1];
ConfigData.rec6_Pusher_Speed_2 := List_of_Recipes[6].Pusher.Speed[2];
ConfigData.rec6_Pusher_Speed_3 := List_of_Recipes[6].Pusher.Speed[3];
ConfigData.rec6_Pusher_Speed_4 := List_of_Recipes[6].Pusher.Speed[4];
ConfigData.rec6_Pusher_Speed_5 := List_of_Recipes[6].Pusher.Speed[5];
ConfigData.rec6_Pusher_Speed_6 := List_of_Recipes[6].Pusher.Speed[6];
ConfigData.rec6_Pusher_distance_1 := List_of_Recipes[6].Pusher.distance[1];
ConfigData.rec6_Pusher_distance_2 := List_of_Recipes[6].Pusher.distance[2];
ConfigData.rec6_Pusher_distance_3 := List_of_Recipes[6].Pusher.distance[3];
ConfigData.rec6_Pusher_distance_4 := List_of_Recipes[6].Pusher.distance[4];
ConfigData.rec6_Pusher_distance_5 := List_of_Recipes[6].Pusher.distance[5];
ConfigData.rec6_Pusher_distance_6 := List_of_Recipes[6].Pusher.distance[6];

ConfigData.rec6_Compress_Initial_Distance:= List_of_Recipes[6].Compress.Initial_Distance;
ConfigData.rec6_Compress_Initial_Speed:= List_of_Recipes[6].Compress.Initial_Speed;
ConfigData.rec6_Compress_Relax_Distance:=List_of_Recipes[6].Compress.Relax_Distance;
ConfigData.rec6_Compress_Retract_Speed:=List_of_Recipes[6].Compress.Retract_Speed;

ConfigData.rec6_Clamp_Release_Instance:=List_of_Recipes[6].Clamp.Release_Instance;

ConfigData.rec6_Other_Compress_Home_Offset:=List_of_Recipes[6].Other.Compress_Home_Offset;
ConfigData.rec6_Other_Shield_Home_Offset:=List_of_Recipes[6].Other.Shield_Home_Offset;
ConfigData.rec6_Other_Pusher_Home_Offset:=List_of_Recipes[6].Other.Pusher_Home_Offset;

ConfigData.rec6_Memory_Free:=BOOL_TO_LREAL(List_of_Recipes[6].Memory_Free);


//7


Recipe_mem_name := List_of_Recipes[7].Name;

ConfigData.rec7_Name_1:=Rec_Name_1;								
ConfigData.rec7_Name_2:=Rec_Name_2;								
ConfigData.rec7_Name_3:=Rec_Name_3;								
ConfigData.rec7_Name_4:=Rec_Name_4;								
ConfigData.rec7_Name_5:=Rec_Name_5;

ConfigData.rec7_Shield_Retract_Speed := List_of_Recipes[7].Shield.Retract_Speed;
ConfigData.rec7_Shield_Speed_1 := List_of_Recipes[7].Shield.Speed[1];
ConfigData.rec7_Shield_Speed_2 := List_of_Recipes[7].Shield.Speed[2];
ConfigData.rec7_Shield_Speed_3 := List_of_Recipes[7].Shield.Speed[3];
ConfigData.rec7_Shield_Speed_4 := List_of_Recipes[7].Shield.Speed[4];
ConfigData.rec7_Shield_Speed_5 := List_of_Recipes[7].Shield.Speed[5];
ConfigData.rec7_Shield_Speed_6 := List_of_Recipes[7].Shield.Speed[6];
ConfigData.rec7_Shield_distance_1 := List_of_Recipes[7].Shield.distance[1];
ConfigData.rec7_Shield_distance_2 := List_of_Recipes[7].Shield.distance[2];
ConfigData.rec7_Shield_distance_3 := List_of_Recipes[7].Shield.distance[3];
ConfigData.rec7_Shield_distance_4 := List_of_Recipes[7].Shield.distance[4];
ConfigData.rec7_Shield_distance_5 := List_of_Recipes[7].Shield.distance[5];
ConfigData.rec7_Shield_distance_6 := List_of_Recipes[7].Shield.distance[6];


ConfigData.rec7_Pusher_Retract_Speed := List_of_Recipes[7].Pusher.Retract_Speed;
ConfigData.rec7_Pusher_Speed_1 := List_of_Recipes[7].Pusher.Speed[1];
ConfigData.rec7_Pusher_Speed_2 := List_of_Recipes[7].Pusher.Speed[2];
ConfigData.rec7_Pusher_Speed_3 := List_of_Recipes[7].Pusher.Speed[3];
ConfigData.rec7_Pusher_Speed_4 := List_of_Recipes[7].Pusher.Speed[4];
ConfigData.rec7_Pusher_Speed_5 := List_of_Recipes[7].Pusher.Speed[5];
ConfigData.rec7_Pusher_Speed_6 := List_of_Recipes[7].Pusher.Speed[6];
ConfigData.rec7_Pusher_distance_1 := List_of_Recipes[7].Pusher.distance[1];
ConfigData.rec7_Pusher_distance_2 := List_of_Recipes[7].Pusher.distance[2];
ConfigData.rec7_Pusher_distance_3 := List_of_Recipes[7].Pusher.distance[3];
ConfigData.rec7_Pusher_distance_4 := List_of_Recipes[7].Pusher.distance[4];
ConfigData.rec7_Pusher_distance_5 := List_of_Recipes[7].Pusher.distance[5];
ConfigData.rec7_Pusher_distance_6 := List_of_Recipes[7].Pusher.distance[6];

ConfigData.rec7_Compress_Initial_Distance:= List_of_Recipes[7].Compress.Initial_Distance;
ConfigData.rec7_Compress_Initial_Speed:= List_of_Recipes[7].Compress.Initial_Speed;
ConfigData.rec7_Compress_Relax_Distance:=List_of_Recipes[7].Compress.Relax_Distance;
ConfigData.rec7_Compress_Retract_Speed:=List_of_Recipes[7].Compress.Retract_Speed;

ConfigData.rec7_Clamp_Release_Instance:=List_of_Recipes[7].Clamp.Release_Instance;

ConfigData.rec7_Other_Compress_Home_Offset:=List_of_Recipes[7].Other.Compress_Home_Offset;
ConfigData.rec7_Other_Shield_Home_Offset:=List_of_Recipes[7].Other.Shield_Home_Offset;
ConfigData.rec7_Other_Pusher_Home_Offset:=List_of_Recipes[7].Other.Pusher_Home_Offset;

ConfigData.rec7_Memory_Free:=BOOL_TO_LREAL(List_of_Recipes[7].Memory_Free);

//8


Recipe_mem_name := List_of_Recipes[8].Name;

ConfigData.rec8_Name_1:=Rec_Name_1;								
ConfigData.rec8_Name_2:=Rec_Name_2;								
ConfigData.rec8_Name_3:=Rec_Name_3;								
ConfigData.rec8_Name_4:=Rec_Name_4;								
ConfigData.rec8_Name_5:=Rec_Name_5;

ConfigData.rec8_Shield_Retract_Speed := List_of_Recipes[8].Shield.Retract_Speed;
ConfigData.rec8_Shield_Speed_1 := List_of_Recipes[8].Shield.Speed[1];
ConfigData.rec8_Shield_Speed_2 := List_of_Recipes[8].Shield.Speed[2];
ConfigData.rec8_Shield_Speed_3 := List_of_Recipes[8].Shield.Speed[3];
ConfigData.rec8_Shield_Speed_4 := List_of_Recipes[8].Shield.Speed[4];
ConfigData.rec8_Shield_Speed_5 := List_of_Recipes[8].Shield.Speed[5];
ConfigData.rec8_Shield_Speed_6 := List_of_Recipes[8].Shield.Speed[6];
ConfigData.rec8_Shield_distance_1 := List_of_Recipes[8].Shield.distance[1];
ConfigData.rec8_Shield_distance_2 := List_of_Recipes[8].Shield.distance[2];
ConfigData.rec8_Shield_distance_3 := List_of_Recipes[8].Shield.distance[3];
ConfigData.rec8_Shield_distance_4 := List_of_Recipes[8].Shield.distance[4];
ConfigData.rec8_Shield_distance_5 := List_of_Recipes[8].Shield.distance[5];
ConfigData.rec8_Shield_distance_6 := List_of_Recipes[8].Shield.distance[6];


ConfigData.rec8_Pusher_Retract_Speed := List_of_Recipes[8].Pusher.Retract_Speed;
ConfigData.rec8_Pusher_Speed_1 := List_of_Recipes[8].Pusher.Speed[1];
ConfigData.rec8_Pusher_Speed_2 := List_of_Recipes[8].Pusher.Speed[2];
ConfigData.rec8_Pusher_Speed_3 := List_of_Recipes[8].Pusher.Speed[3];
ConfigData.rec8_Pusher_Speed_4 := List_of_Recipes[8].Pusher.Speed[4];
ConfigData.rec8_Pusher_Speed_5 := List_of_Recipes[8].Pusher.Speed[5];
ConfigData.rec8_Pusher_Speed_6 := List_of_Recipes[8].Pusher.Speed[6];
ConfigData.rec8_Pusher_distance_1 := List_of_Recipes[8].Pusher.distance[1];
ConfigData.rec8_Pusher_distance_2 := List_of_Recipes[8].Pusher.distance[2];
ConfigData.rec8_Pusher_distance_3 := List_of_Recipes[8].Pusher.distance[3];
ConfigData.rec8_Pusher_distance_4 := List_of_Recipes[8].Pusher.distance[4];
ConfigData.rec8_Pusher_distance_5 := List_of_Recipes[8].Pusher.distance[5];
ConfigData.rec8_Pusher_distance_6 := List_of_Recipes[8].Pusher.distance[6];

ConfigData.rec8_Compress_Initial_Distance:= List_of_Recipes[8].Compress.Initial_Distance;
ConfigData.rec8_Compress_Initial_Speed:= List_of_Recipes[8].Compress.Initial_Speed;
ConfigData.rec8_Compress_Relax_Distance:=List_of_Recipes[8].Compress.Relax_Distance;
ConfigData.rec8_Compress_Retract_Speed:=List_of_Recipes[8].Compress.Retract_Speed;

ConfigData.rec8_Clamp_Release_Instance:=List_of_Recipes[8].Clamp.Release_Instance;

ConfigData.rec8_Other_Compress_Home_Offset:=List_of_Recipes[8].Other.Compress_Home_Offset;
ConfigData.rec8_Other_Shield_Home_Offset:=List_of_Recipes[8].Other.Shield_Home_Offset;
ConfigData.rec8_Other_Pusher_Home_Offset:=List_of_Recipes[8].Other.Pusher_Home_Offset;

ConfigData.rec8_Memory_Free:=BOOL_TO_LREAL(List_of_Recipes[8].Memory_Free);

//9


Recipe_mem_name := List_of_Recipes[9].Name;

ConfigData.rec9_Name_1:=Rec_Name_1;								
ConfigData.rec9_Name_2:=Rec_Name_2;								
ConfigData.rec9_Name_3:=Rec_Name_3;								
ConfigData.rec9_Name_4:=Rec_Name_4;								
ConfigData.rec9_Name_5:=Rec_Name_5;

ConfigData.rec9_Shield_Retract_Speed := List_of_Recipes[9].Shield.Retract_Speed;
ConfigData.rec9_Shield_Speed_1 := List_of_Recipes[9].Shield.Speed[1];
ConfigData.rec9_Shield_Speed_2 := List_of_Recipes[9].Shield.Speed[2];
ConfigData.rec9_Shield_Speed_3 := List_of_Recipes[9].Shield.Speed[3];
ConfigData.rec9_Shield_Speed_4 := List_of_Recipes[9].Shield.Speed[4];
ConfigData.rec9_Shield_Speed_5 := List_of_Recipes[9].Shield.Speed[5];
ConfigData.rec9_Shield_Speed_6 := List_of_Recipes[9].Shield.Speed[6];
ConfigData.rec9_Shield_distance_1 := List_of_Recipes[9].Shield.distance[1];
ConfigData.rec9_Shield_distance_2 := List_of_Recipes[9].Shield.distance[2];
ConfigData.rec9_Shield_distance_3 := List_of_Recipes[9].Shield.distance[3];
ConfigData.rec9_Shield_distance_4 := List_of_Recipes[9].Shield.distance[4];
ConfigData.rec9_Shield_distance_5 := List_of_Recipes[9].Shield.distance[5];
ConfigData.rec9_Shield_distance_6 := List_of_Recipes[9].Shield.distance[6];


ConfigData.rec9_Pusher_Retract_Speed := List_of_Recipes[9].Pusher.Retract_Speed;
ConfigData.rec9_Pusher_Speed_1 := List_of_Recipes[9].Pusher.Speed[1];
ConfigData.rec9_Pusher_Speed_2 := List_of_Recipes[9].Pusher.Speed[2];
ConfigData.rec9_Pusher_Speed_3 := List_of_Recipes[9].Pusher.Speed[3];
ConfigData.rec9_Pusher_Speed_4 := List_of_Recipes[9].Pusher.Speed[4];
ConfigData.rec9_Pusher_Speed_5 := List_of_Recipes[9].Pusher.Speed[5];
ConfigData.rec9_Pusher_Speed_6 := List_of_Recipes[9].Pusher.Speed[6];
ConfigData.rec9_Pusher_distance_1 := List_of_Recipes[9].Pusher.distance[1];
ConfigData.rec9_Pusher_distance_2 := List_of_Recipes[9].Pusher.distance[2];
ConfigData.rec9_Pusher_distance_3 := List_of_Recipes[9].Pusher.distance[3];
ConfigData.rec9_Pusher_distance_4 := List_of_Recipes[9].Pusher.distance[4];
ConfigData.rec9_Pusher_distance_5 := List_of_Recipes[9].Pusher.distance[5];
ConfigData.rec9_Pusher_distance_6 := List_of_Recipes[9].Pusher.distance[6];

ConfigData.rec9_Compress_Initial_Distance:= List_of_Recipes[9].Compress.Initial_Distance;
ConfigData.rec9_Compress_Initial_Speed:= List_of_Recipes[9].Compress.Initial_Speed;
ConfigData.rec9_Compress_Relax_Distance:=List_of_Recipes[9].Compress.Relax_Distance;
ConfigData.rec9_Compress_Retract_Speed:=List_of_Recipes[9].Compress.Retract_Speed;

ConfigData.rec9_Clamp_Release_Instance:=List_of_Recipes[9].Clamp.Release_Instance;

ConfigData.rec9_Other_Compress_Home_Offset:=List_of_Recipes[9].Other.Compress_Home_Offset;
ConfigData.rec9_Other_Shield_Home_Offset:=List_of_Recipes[9].Other.Shield_Home_Offset;
ConfigData.rec9_Other_Pusher_Home_Offset:=List_of_Recipes[9].Other.Pusher_Home_Offset;

ConfigData.rec9_Memory_Free:=BOOL_TO_LREAL(List_of_Recipes[9].Memory_Free);

//10


Recipe_mem_name := List_of_Recipes[10].Name;

ConfigData.rec10_Name_1:=Rec_Name_1;								
ConfigData.rec10_Name_2:=Rec_Name_2;								
ConfigData.rec10_Name_3:=Rec_Name_3;								
ConfigData.rec10_Name_4:=Rec_Name_4;								
ConfigData.rec10_Name_5:=Rec_Name_5;

ConfigData.rec10_Shield_Retract_Speed := List_of_Recipes[10].Shield.Retract_Speed;
ConfigData.rec10_Shield_Speed_1 := List_of_Recipes[10].Shield.Speed[1];
ConfigData.rec10_Shield_Speed_2 := List_of_Recipes[10].Shield.Speed[2];
ConfigData.rec10_Shield_Speed_3 := List_of_Recipes[10].Shield.Speed[3];
ConfigData.rec10_Shield_Speed_4 := List_of_Recipes[10].Shield.Speed[4];
ConfigData.rec10_Shield_Speed_5 := List_of_Recipes[10].Shield.Speed[5];
ConfigData.rec10_Shield_Speed_6 := List_of_Recipes[10].Shield.Speed[6];
ConfigData.rec10_Shield_distance_1 := List_of_Recipes[10].Shield.distance[1];
ConfigData.rec10_Shield_distance_2 := List_of_Recipes[10].Shield.distance[2];
ConfigData.rec10_Shield_distance_3 := List_of_Recipes[10].Shield.distance[3];
ConfigData.rec10_Shield_distance_4 := List_of_Recipes[10].Shield.distance[4];
ConfigData.rec10_Shield_distance_5 := List_of_Recipes[10].Shield.distance[5];
ConfigData.rec10_Shield_distance_6 := List_of_Recipes[10].Shield.distance[6];


ConfigData.rec10_Pusher_Retract_Speed := List_of_Recipes[10].Pusher.Retract_Speed;
ConfigData.rec10_Pusher_Speed_1 := List_of_Recipes[10].Pusher.Speed[1];
ConfigData.rec10_Pusher_Speed_2 := List_of_Recipes[10].Pusher.Speed[2];
ConfigData.rec10_Pusher_Speed_3 := List_of_Recipes[10].Pusher.Speed[3];
ConfigData.rec10_Pusher_Speed_4 := List_of_Recipes[10].Pusher.Speed[4];
ConfigData.rec10_Pusher_Speed_5 := List_of_Recipes[10].Pusher.Speed[5];
ConfigData.rec10_Pusher_Speed_6 := List_of_Recipes[10].Pusher.Speed[6];
ConfigData.rec10_Pusher_distance_1 := List_of_Recipes[10].Pusher.distance[1];
ConfigData.rec10_Pusher_distance_2 := List_of_Recipes[10].Pusher.distance[2];
ConfigData.rec10_Pusher_distance_3 := List_of_Recipes[10].Pusher.distance[3];
ConfigData.rec10_Pusher_distance_4 := List_of_Recipes[10].Pusher.distance[4];
ConfigData.rec10_Pusher_distance_5 := List_of_Recipes[10].Pusher.distance[5];
ConfigData.rec10_Pusher_distance_6 := List_of_Recipes[10].Pusher.distance[6];

ConfigData.rec10_Compress_Initial_Distance:= List_of_Recipes[10].Compress.Initial_Distance;
ConfigData.rec10_Compress_Initial_Speed:= List_of_Recipes[10].Compress.Initial_Speed;
ConfigData.rec10_Compress_Relax_Distance:=List_of_Recipes[10].Compress.Relax_Distance;
ConfigData.rec10_Compress_Retract_Speed:=List_of_Recipes[10].Compress.Retract_Speed;

ConfigData.rec10_Clamp_Release_Instance:=List_of_Recipes[10].Clamp.Release_Instance;

ConfigData.rec10_Other_Compress_Home_Offset:=List_of_Recipes[10].Other.Compress_Home_Offset;
ConfigData.rec10_Other_Shield_Home_Offset:=List_of_Recipes[10].Other.Shield_Home_Offset;
ConfigData.rec10_Other_Pusher_Home_Offset:=List_of_Recipes[10].Other.Pusher_Home_Offset;

ConfigData.rec10_Memory_Free:=BOOL_TO_LREAL(List_of_Recipes[10].Memory_Free);
END_METHOD

METHOD Initialised : BOOL
VAR_INPUT

END_VAR
Initialised := ConfigData.Initialised;
END_METHOD

METHOD Update : BOOL
VAR_INPUT
	
	
END_VAR
VAR
	recipe_file_name			:STRING;
	ThisErrrorId				: UDINT;
	ThisErrorText				: STRING;
	ThisError					: BOOL;
END_VAR

recipe_file_name:='Hard Disk\TwinCAT\3.1\Boot\all_recipes_limits';

PersistentData(
	//DataAddress:= ADR(ConfigData[save_load_no_u]), 
	//DataLength:= SIZEOF(ConfigData[save_load_no_u]), 
	DataAddress:= ADR(ConfigData), 
	DataLength:= SIZEOF(ConfigData), 
	Filename:= recipe_file_name, 
	Timestamp:= Clock.DateTimeAsString, 
	LoadFromFile:= NOT ConfigData.Initialised, 
	AutoSave:= TRUE, 
	ValuesReadFromFile=> ConfigData.Initialised, 
	Error=>ThisError , 
	ErrorId=> ThisErrrorId, 
	ErrorText=>ThisErrorText );
	
IF (ThisError) THEN
	ThisErrrorId:=ThisErrrorId;
END_IF
END_METHOD

END_FUNCTION_BLOCK

// ---- POUs/F_DisplayText.TcPOU
FUNCTION F_DisplayText : STRING
VAR_INPUT
	InputString: WSTRING;
	InputNumber: WORD;
END_VAR
VAR
	Text : STRING;
	Join : STRING;
	TextPlus : STRING;
	number : STRING;
END_VAR

Text := WSTRING_TO_STRING(InputString);
Number := WORD_TO_STRING(InputNumber);
IF InputNumber = 0 THEN
	F_DisplayText := Text;
ELSE
	Join := WSTRING_TO_STRING(" #");
	TextPlus := concat(Text,Join);
	F_DisplayText := concat(TextPlus,Number);
END_IF

END_FUNCTION

// ---- XML/FB_RetainedData.TcPOU
FUNCTION_BLOCK FB_RetainedData
VAR_INPUT
	xSaveAll								: BOOL;
END_VAR
VAR_OUTPUT
	xReadComplete							: BOOL;
	xErr									: BOOL;
	nErrID									: UDINT;
	RecipeSaveDone: BOOL;
END_VAR
VAR
	//fbRetainGlobalSettings					: FB_Retain;
	fbRetainRecipes							: FB_Retain;
	
	xAllRead								: BOOL;
	tonFileReadComplete						: ton;
	testbit: BOOL;
END_VAR

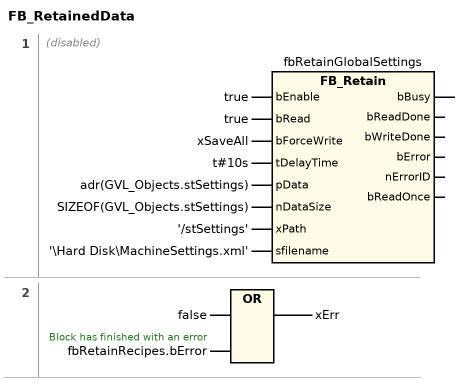
// NETWORK 1 (disabled)
// fbRetainGlobalSettings(
//     bEnable := true,
//     bRead := true,
//     bForceWrite := xSaveAll,
//     tDelayTime := t#10s,
//     pData := adr(GVL_Objects.stSettings),
//     nDataSize := SIZEOF(GVL_Objects.stSettings),
//     xPath := '/stSettings',
//     sfilename := '\Hard Disk\MachineSettings.xml'); // FB_Retain

// NETWORK 2
//   fbRetainRecipes.bError: Block has finished with an error
xErr := false OR fbRetainRecipes.bError;

END_FUNCTION_BLOCK
